Yaskawa INFORM job: A_ROOF_UPPER_0614_2_PAINT_13.JBI

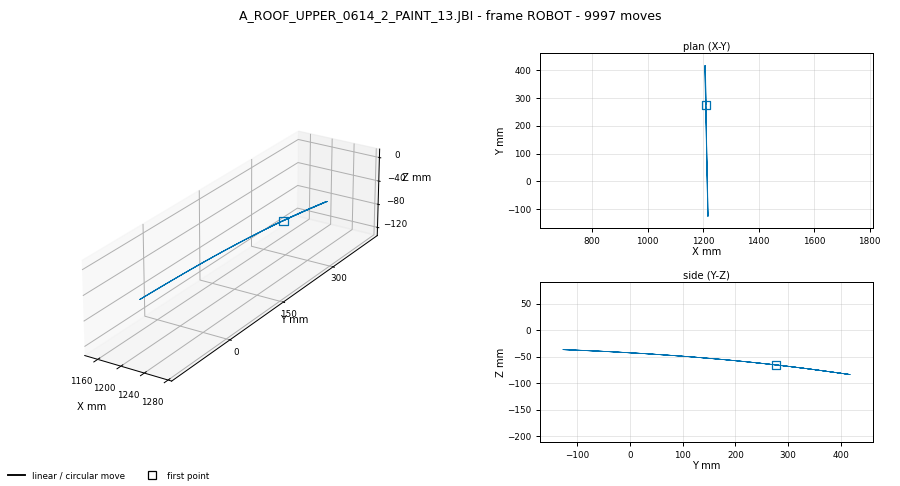
[picture p0: tool path of A_ROOF_UPPER_0614_2_PAINT_13.JBI in frame ROBOT, 9997 of 9997 moves have a stored position in this frame; points joined in program order, loops and branches not executed]
/JOB
//NAME A_ROOF_UPPER_0614_2_PAINT13
//POS
///NPOS 9997,0,0,0,0,0
///TOOL 1
///USER 0
///POSTYPE ROBOT
///RECTAN
///RCONF 1,0,0,0,0,0,0,0,0,0,0,0,0,0,0,0,0,0,0,0,0,0,0,0
C00000=1210.208,276.107,-65.224,-176.767,6.904,148.334
C00001=1210.203,276.355,-65.252,-176.765,6.906,148.334
C00002=1210.199,276.604,-65.280,-176.762,6.909,148.334
C00003=1210.195,276.851,-65.308,-176.760,6.911,148.334
C00004=1210.190,277.100,-65.337,-176.757,6.914,148.333
C00005=1210.186,277.348,-65.365,-176.754,6.916,148.333
C00006=1210.182,277.597,-65.393,-176.752,6.918,148.333
C00007=1210.177,277.845,-65.421,-176.749,6.921,148.333
C00008=1210.173,278.093,-65.449,-176.747,6.923,148.333
C00009=1210.169,278.342,-65.478,-176.744,6.926,148.333
C00010=1210.164,278.590,-65.506,-176.742,6.928,148.333
C00011=1210.160,278.839,-65.535,-176.740,6.930,148.333
C00012=1210.156,279.087,-65.562,-176.737,6.933,148.333
C00013=1210.151,279.335,-65.592,-176.734,6.935,148.332
C00014=1210.147,279.583,-65.620,-176.732,6.938,148.332
C00015=1210.143,279.832,-65.648,-176.729,6.940,148.332
C00016=1210.138,280.080,-65.676,-176.727,6.942,148.332
C00017=1210.134,280.329,-65.705,-176.724,6.945,148.332
C00018=1210.129,280.577,-65.733,-176.722,6.947,148.332
C00019=1210.125,280.826,-65.761,-176.719,6.950,148.332
C00020=1210.121,281.074,-65.790,-176.717,6.952,148.331
C00021=1210.116,281.322,-65.819,-176.715,6.955,148.331
C00022=1210.113,281.570,-65.847,-176.712,6.958,148.331
C00023=1210.107,281.818,-65.875,-176.709,6.959,148.331
C00024=1210.104,282.067,-65.903,-176.707,6.962,148.331
C00025=1210.099,282.316,-65.932,-176.704,6.965,148.331
C00026=1210.094,282.564,-65.961,-176.701,6.967,148.331
C00027=1210.091,282.812,-65.989,-176.699,6.970,148.331
C00028=1210.086,283.060,-66.018,-176.697,6.972,148.331
C00029=1210.082,283.308,-66.047,-176.694,6.975,148.331
C00030=1210.078,283.557,-66.075,-176.692,6.977,148.330
C00031=1210.073,283.805,-66.104,-176.689,6.980,148.330
C00032=1210.069,284.054,-66.132,-176.687,6.982,148.330
C00033=1210.064,284.301,-66.161,-176.685,6.984,148.330
C00034=1210.060,284.550,-66.190,-176.682,6.987,148.330
C00035=1210.056,284.799,-66.218,-176.679,6.989,148.330
C00036=1210.051,285.046,-66.247,-176.677,6.992,148.330
C00037=1210.047,285.295,-66.276,-176.675,6.994,148.330
C00038=1210.043,285.544,-66.304,-176.672,6.997,148.329
C00039=1210.038,285.791,-66.333,-176.669,6.999,148.329
C00040=1210.034,286.040,-66.362,-176.667,7.002,148.329
C00041=1210.030,286.288,-66.390,-176.665,7.004,148.329
C00042=1210.025,286.537,-66.419,-176.662,7.006,148.329
C00043=1210.021,286.785,-66.448,-176.659,7.009,148.329
C00044=1210.016,287.034,-66.477,-176.657,7.011,148.329
C00045=1210.012,287.282,-66.505,-176.654,7.014,148.329
C00046=1210.008,287.530,-66.534,-176.652,7.016,148.329
C00047=1210.003,287.779,-66.563,-176.649,7.019,148.329
C00048=1209.999,288.026,-66.592,-176.647,7.022,148.329
C00049=1209.995,288.275,-66.620,-176.644,7.025,148.329
C00050=1209.991,288.523,-66.650,-176.642,7.027,148.328
C00051=1209.986,288.797,-66.681,-176.639,7.030,148.328
C00052=1209.981,289.071,-66.714,-176.636,7.033,148.328
C00053=1209.977,289.346,-66.745,-176.634,7.036,148.328
C00054=1209.971,289.620,-66.778,-176.631,7.037,148.328
C00055=1209.968,289.868,-66.806,-176.628,7.040,148.328
C00056=1209.963,290.117,-66.835,-176.626,7.043,148.328
C00057=1209.958,290.365,-66.864,-176.624,7.046,148.328
C00058=1209.954,290.613,-66.894,-176.621,7.048,148.328
C00059=1209.950,290.862,-66.922,-176.618,7.051,148.327
C00060=1209.945,291.110,-66.952,-176.616,7.053,148.327
C00061=1209.941,291.357,-66.980,-176.614,7.056,148.327
C00062=1209.937,291.606,-67.009,-176.611,7.058,148.327
C00063=1209.933,291.854,-67.039,-176.609,7.061,148.327
C00064=1209.929,292.103,-67.068,-176.607,7.063,148.327
C00065=1209.924,292.352,-67.097,-176.603,7.066,148.327
C00066=1209.919,292.599,-67.126,-176.601,7.068,148.327
C00067=1209.915,292.847,-67.155,-176.599,7.070,148.327
C00068=1209.911,293.096,-67.184,-176.596,7.073,148.327
C00069=1209.906,293.345,-67.213,-176.594,7.076,148.327
C00070=1209.902,293.593,-67.243,-176.592,7.079,148.327
C00071=1209.897,293.840,-67.272,-176.590,7.081,148.327
C00072=1209.894,294.088,-67.301,-176.586,7.084,148.326
C00073=1209.889,294.337,-67.330,-176.584,7.086,148.326
C00074=1209.885,294.586,-67.359,-176.582,7.089,148.326
C00075=1209.881,294.834,-67.388,-176.579,7.091,148.326
C00076=1209.876,295.081,-67.418,-176.577,7.094,148.326
C00077=1209.872,295.330,-67.447,-176.575,7.096,148.326
C00078=1209.868,295.578,-67.476,-176.572,7.099,148.326
C00079=1209.864,295.826,-67.506,-176.570,7.101,148.326
C00080=1209.859,296.075,-67.535,-176.567,7.104,148.326
C00081=1209.855,296.323,-67.564,-176.565,7.106,148.326
C00082=1209.851,296.572,-67.594,-176.562,7.109,148.326
C00083=1209.847,296.820,-67.623,-176.560,7.112,148.326
C00084=1209.842,297.067,-67.652,-176.557,7.115,148.326
C00085=1209.838,297.316,-67.682,-176.555,7.117,148.326
C00086=1209.834,297.564,-67.711,-176.552,7.120,148.326
C00087=1209.829,297.813,-67.741,-176.550,7.122,148.326
C00088=1209.825,298.061,-67.771,-176.547,7.125,148.326
C00089=1209.820,298.309,-67.800,-176.545,7.127,148.326
C00090=1209.816,298.557,-67.829,-176.543,7.130,148.326
C00091=1209.812,298.806,-67.859,-176.540,7.132,148.325
C00092=1209.808,299.054,-67.888,-176.537,7.135,148.325
C00093=1209.804,299.302,-67.918,-176.535,7.137,148.325
C00094=1209.799,299.550,-67.947,-176.533,7.140,148.325
C00095=1209.795,299.798,-67.976,-176.530,7.143,148.325
C00096=1209.790,300.046,-68.006,-176.528,7.146,148.325
C00097=1209.786,300.295,-68.036,-176.526,7.148,148.325
C00098=1209.782,300.543,-68.066,-176.523,7.151,148.325
C00099=1209.777,300.791,-68.095,-176.521,7.153,148.325
C00100=1209.773,301.039,-68.125,-176.518,7.156,148.325
C00101=1209.769,301.287,-68.154,-176.515,7.159,148.325
C00102=1209.765,301.536,-68.184,-176.513,7.161,148.325
C00103=1209.760,301.784,-68.214,-176.511,7.164,148.325
C00104=1209.756,302.032,-68.243,-176.508,7.167,148.325
C00105=1209.752,302.280,-68.273,-176.506,7.170,148.325
C00106=1209.748,302.528,-68.303,-176.504,7.172,148.325
C00107=1209.743,302.777,-68.333,-176.501,7.175,148.325
C00108=1209.739,303.025,-68.362,-176.499,7.177,148.325
C00109=1209.735,303.273,-68.392,-176.496,7.180,148.325
C00110=1209.731,303.521,-68.422,-176.494,7.182,148.325
C00111=1209.726,303.770,-68.452,-176.491,7.185,148.325
C00112=1209.722,304.018,-68.482,-176.489,7.188,148.324
C00113=1209.718,304.266,-68.512,-176.487,7.191,148.324
C00114=1209.713,304.514,-68.541,-176.484,7.193,148.324
C00115=1209.709,304.762,-68.571,-176.482,7.196,148.324
C00116=1209.704,305.011,-68.601,-176.480,7.198,148.324
C00117=1209.700,305.258,-68.631,-176.477,7.201,148.324
C00118=1209.696,305.507,-68.661,-176.474,7.204,148.324
C00119=1209.692,305.755,-68.691,-176.472,7.206,148.324
C00120=1209.688,306.003,-68.721,-176.469,7.209,148.324
C00121=1209.683,306.251,-68.751,-176.467,7.211,148.324
C00122=1209.679,306.499,-68.781,-176.465,7.215,148.324
C00123=1209.675,306.747,-68.810,-176.463,7.217,148.324
C00124=1209.670,306.995,-68.841,-176.460,7.220,148.324
C00125=1209.666,307.244,-68.870,-176.458,7.222,148.324
C00126=1209.662,307.492,-68.900,-176.456,7.225,148.324
C00127=1209.657,307.740,-68.931,-176.453,7.227,148.324
C00128=1209.653,307.988,-68.960,-176.451,7.231,148.324
C00129=1209.649,308.237,-68.991,-176.448,7.234,148.324
C00130=1209.645,308.485,-69.021,-176.446,7.236,148.324
C00131=1209.641,308.733,-69.051,-176.443,7.239,148.324
C00132=1209.636,308.981,-69.081,-176.441,7.241,148.324
C00133=1209.632,309.229,-69.111,-176.438,7.244,148.324
C00134=1209.627,309.477,-69.141,-176.436,7.246,148.324
C00135=1209.623,309.725,-69.171,-176.434,7.249,148.324
C00136=1209.618,309.973,-69.202,-176.432,7.252,148.324
C00137=1209.614,310.221,-69.232,-176.429,7.255,148.324
C00138=1209.610,310.469,-69.262,-176.427,7.257,148.324
C00139=1209.606,310.718,-69.292,-176.425,7.260,148.324
C00140=1209.602,310.966,-69.322,-176.422,7.263,148.324
C00141=1209.598,311.214,-69.353,-176.420,7.265,148.324
C00142=1209.593,311.462,-69.382,-176.417,7.268,148.324
C00143=1209.589,311.710,-69.413,-176.415,7.271,148.324
C00144=1209.585,311.958,-69.443,-176.413,7.274,148.324
C00145=1209.580,312.206,-69.473,-176.411,7.276,148.324
C00146=1209.577,312.455,-69.504,-176.408,7.279,148.324
C00147=1209.572,312.703,-69.535,-176.406,7.281,148.324
C00148=1209.567,312.951,-69.565,-176.403,7.284,148.324
C00149=1209.563,313.199,-69.595,-176.400,7.287,148.324
C00150=1209.559,313.447,-69.626,-176.399,7.290,148.324
C00151=1209.555,313.696,-69.656,-176.396,7.293,148.324
C00152=1209.551,313.944,-69.686,-176.394,7.295,148.324
C00153=1209.547,314.191,-69.716,-176.391,7.298,148.324
C00154=1209.542,314.439,-69.747,-176.389,7.300,148.324
C00155=1209.537,314.716,-69.781,-176.387,7.303,148.324
C00156=1209.532,314.992,-69.815,-176.384,7.307,148.324
C00157=1209.528,315.268,-69.848,-176.382,7.310,148.324
C00158=1209.524,315.544,-69.883,-176.379,7.313,148.324
C00159=1209.519,315.792,-69.913,-176.376,7.316,148.324
C00160=1209.514,316.040,-69.944,-176.374,7.318,148.324
C00161=1209.511,316.288,-69.974,-176.372,7.321,148.324
C00162=1209.506,316.536,-70.005,-176.369,7.324,148.324
C00163=1209.502,316.785,-70.036,-176.367,7.327,148.324
C00164=1209.498,317.033,-70.066,-176.364,7.330,148.324
C00165=1209.493,317.281,-70.097,-176.362,7.332,148.324
C00166=1209.489,317.529,-70.128,-176.360,7.335,148.325
C00167=1209.485,317.777,-70.158,-176.358,7.337,148.325
C00168=1209.481,318.025,-70.189,-176.355,7.340,148.325
C00169=1209.476,318.273,-70.219,-176.353,7.344,148.325
C00170=1209.473,318.521,-70.250,-176.351,7.346,148.325
C00171=1209.468,318.769,-70.281,-176.348,7.349,148.325
C00172=1209.464,319.017,-70.311,-176.346,7.351,148.325
C00173=1209.459,319.265,-70.342,-176.344,7.355,148.325
C00174=1209.456,319.513,-70.373,-176.342,7.357,148.325
C00175=1209.451,319.761,-70.403,-176.339,7.360,148.325
C00176=1209.446,320.009,-70.434,-176.337,7.363,148.325
C00177=1209.442,320.258,-70.465,-176.335,7.365,148.325
C00178=1209.439,320.506,-70.496,-176.332,7.368,148.325
C00179=1209.434,320.753,-70.527,-176.331,7.371,148.325
C00180=1209.430,321.002,-70.558,-176.328,7.374,148.325
C00181=1209.426,321.249,-70.589,-176.325,7.377,148.325
C00182=1209.422,321.497,-70.619,-176.324,7.380,148.325
C00183=1209.418,321.746,-70.650,-176.321,7.383,148.325
C00184=1209.413,321.994,-70.681,-176.319,7.385,148.325
C00185=1209.408,322.242,-70.712,-176.317,7.388,148.325
C00186=1209.405,322.490,-70.744,-176.314,7.390,148.325
C00187=1209.400,322.738,-70.774,-176.312,7.393,148.325
C00188=1209.396,322.985,-70.805,-176.310,7.397,148.326
C00189=1209.392,323.234,-70.836,-176.307,7.399,148.326
C00190=1209.388,323.482,-70.866,-176.305,7.402,148.326
C00191=1209.384,323.730,-70.898,-176.303,7.404,148.326
C00192=1209.379,323.978,-70.929,-176.300,7.408,148.326
C00193=1209.375,324.226,-70.960,-176.299,7.410,148.326
C00194=1209.371,324.475,-70.991,-176.296,7.413,148.326
C00195=1209.366,324.722,-71.022,-176.293,7.416,148.326
C00196=1209.363,324.970,-71.053,-176.292,7.419,148.326
C00197=1209.359,325.218,-71.084,-176.289,7.422,148.326
C00198=1209.354,325.466,-71.115,-176.287,7.424,148.326
C00199=1209.350,325.714,-71.146,-176.285,7.427,148.326
C00200=1209.346,325.962,-71.177,-176.283,7.431,148.326
C00201=1209.342,326.210,-71.209,-176.280,7.433,148.326
C00202=1209.337,326.458,-71.240,-176.278,7.436,148.326
C00203=1209.333,326.707,-71.271,-176.276,7.438,148.327
C00204=1209.329,326.954,-71.302,-176.273,7.441,148.327
C00205=1209.324,327.202,-71.333,-176.272,7.444,148.327
C00206=1209.321,327.450,-71.365,-176.269,7.447,148.327
C00207=1209.316,327.698,-71.396,-176.267,7.450,148.327
C00208=1209.312,327.947,-71.427,-176.265,7.452,148.327
C00209=1209.308,328.194,-71.458,-176.263,7.456,148.327
C00210=1209.304,328.443,-71.489,-176.260,7.458,148.327
C00211=1209.299,328.690,-71.521,-176.258,7.461,148.327
C00212=1209.295,328.939,-71.552,-176.256,7.464,148.327
C00213=1209.291,329.186,-71.583,-176.254,7.467,148.328
C00214=1209.287,329.435,-71.615,-176.251,7.470,148.328
C00215=1209.283,329.682,-71.646,-176.250,7.472,148.328
C00216=1209.279,329.931,-71.677,-176.247,7.475,148.328
C00217=1209.274,330.178,-71.709,-176.245,7.478,148.328
C00218=1209.270,330.427,-71.740,-176.243,7.481,148.328
C00219=1209.265,330.674,-71.772,-176.240,7.484,148.328
C00220=1209.262,330.922,-71.804,-176.238,7.487,148.328
C00221=1209.257,331.170,-71.835,-176.236,7.490,148.328
C00222=1209.253,331.418,-71.866,-176.234,7.492,148.328
C00223=1209.249,331.666,-71.897,-176.232,7.495,148.328
C00224=1209.245,331.914,-71.929,-176.229,7.499,148.329
C00225=1209.241,332.162,-71.960,-176.227,7.501,148.329
C00226=1209.237,332.410,-71.992,-176.225,7.504,148.329
C00227=1209.232,332.658,-72.024,-176.224,7.507,148.329
C00228=1209.228,332.906,-72.055,-176.221,7.510,148.329
C00229=1209.223,333.154,-72.086,-176.219,7.512,148.329
C00230=1209.220,333.402,-72.118,-176.217,7.515,148.329
C00231=1209.215,333.649,-72.150,-176.214,7.519,148.329
C00232=1209.212,333.898,-72.181,-176.213,7.521,148.330
C00233=1209.207,334.146,-72.213,-176.210,7.524,148.330
C00234=1209.203,334.394,-72.245,-176.208,7.527,148.330
C00235=1209.199,334.642,-72.276,-176.206,7.530,148.330
C00236=1209.195,334.889,-72.308,-176.203,7.533,148.330
C00237=1209.190,335.138,-72.340,-176.202,7.536,148.330
C00238=1209.185,335.386,-72.371,-176.200,7.539,148.330
C00239=1209.182,335.634,-72.403,-176.197,7.541,148.330
C00240=1209.178,335.882,-72.435,-176.195,7.545,148.331
C00241=1209.174,336.129,-72.466,-176.194,7.547,148.331
C00242=1209.169,336.378,-72.498,-176.191,7.550,148.331
C00243=1209.165,336.625,-72.530,-176.189,7.554,148.331
C00244=1209.161,336.873,-72.561,-176.187,7.556,148.331
C00245=1209.157,337.122,-72.594,-176.184,7.559,148.331
C00246=1209.152,337.369,-72.625,-176.183,7.562,148.331
C00247=1209.149,337.617,-72.657,-176.181,7.565,148.332
C00248=1209.145,337.865,-72.689,-176.179,7.568,148.332
C00249=1209.140,338.113,-72.721,-176.176,7.571,148.332
C00250=1209.136,338.361,-72.753,-176.174,7.574,148.332
C00251=1209.132,338.609,-72.784,-176.172,7.576,148.332
C00252=1209.127,338.857,-72.816,-176.170,7.580,148.332
C00253=1209.123,339.105,-72.848,-176.168,7.582,148.332
C00254=1209.119,339.352,-72.879,-176.166,7.585,148.333
C00255=1209.115,339.601,-72.912,-176.164,7.588,148.333
C00256=1209.111,339.849,-72.944,-176.162,7.591,148.333
C00257=1209.106,340.096,-72.976,-176.159,7.594,148.333
C00258=1209.102,340.344,-73.008,-176.158,7.597,148.333
C00259=1209.097,340.622,-73.044,-176.155,7.600,148.333
C00260=1209.093,340.901,-73.080,-176.153,7.603,148.334
C00261=1209.088,341.178,-73.116,-176.151,7.607,148.334
C00262=1209.083,341.457,-73.151,-176.148,7.610,148.334
C00263=1209.079,341.705,-73.183,-176.146,7.613,148.334
C00264=1209.076,341.952,-73.216,-176.144,7.616,148.334
C00265=1209.071,342.201,-73.248,-176.142,7.619,148.334
C00266=1209.067,342.448,-73.280,-176.141,7.622,148.335
C00267=1209.063,342.696,-73.312,-176.138,7.625,148.335
C00268=1209.059,342.944,-73.344,-176.136,7.628,148.335
C00269=1209.054,343.192,-73.376,-176.135,7.631,148.335
C00270=1209.050,343.440,-73.408,-176.132,7.634,148.335
C00271=1209.046,343.688,-73.441,-176.130,7.636,148.335
C00272=1209.042,343.936,-73.473,-176.128,7.640,148.336
C00273=1209.037,344.184,-73.505,-176.126,7.642,148.336
C00274=1209.034,344.432,-73.537,-176.124,7.646,148.336
C00275=1209.029,344.680,-73.569,-176.122,7.649,148.336
C00276=1209.026,344.927,-73.602,-176.120,7.651,148.336
C00277=1209.021,345.175,-73.634,-176.118,7.655,148.337
C00278=1209.017,345.423,-73.666,-176.116,7.657,148.337
C00279=1209.013,345.671,-73.698,-176.114,7.661,148.337
C00280=1209.009,345.919,-73.731,-176.113,7.663,148.337
C00281=1209.004,346.166,-73.763,-176.110,7.666,148.337
C00282=1209.000,346.415,-73.795,-176.109,7.669,148.338
C00283=1208.996,346.662,-73.828,-176.106,7.672,148.338
C00284=1208.992,346.911,-73.860,-176.105,7.675,148.338
C00285=1208.988,347.159,-73.892,-176.103,7.678,148.338
C00286=1208.983,347.406,-73.925,-176.100,7.681,148.339
C00287=1208.979,347.654,-73.957,-176.099,7.684,148.339
C00288=1208.975,347.902,-73.989,-176.097,7.687,148.339
C00289=1208.971,348.150,-74.022,-176.095,7.690,148.339
C00290=1208.967,348.398,-74.054,-176.093,7.693,148.339
C00291=1208.963,348.645,-74.087,-176.091,7.696,148.340
C00292=1208.958,348.893,-74.120,-176.089,7.699,148.340
C00293=1208.954,349.141,-74.151,-176.087,7.702,148.340
C00294=1208.950,349.389,-74.185,-176.085,7.705,148.340
C00295=1208.946,349.637,-74.217,-176.083,7.707,148.340
C00296=1208.942,349.885,-74.250,-176.081,7.711,148.341
C00297=1208.937,350.132,-74.282,-176.079,7.714,148.341
C00298=1208.933,350.380,-74.315,-176.078,7.717,148.341
C00299=1208.930,350.628,-74.347,-176.075,7.720,148.341
C00300=1208.925,350.876,-74.380,-176.074,7.723,148.342
C00301=1208.921,351.124,-74.412,-176.072,7.726,148.342
C00302=1208.918,351.372,-74.445,-176.070,7.729,148.342
C00303=1208.913,351.620,-74.477,-176.068,7.732,148.342
C00304=1208.908,351.867,-74.510,-176.066,7.735,148.342
C00305=1208.904,352.115,-74.543,-176.064,7.738,148.343
C00306=1208.901,352.363,-74.575,-176.063,7.741,148.343
C00307=1208.896,352.610,-74.608,-176.060,7.744,148.343
C00308=1208.892,352.859,-74.641,-176.059,7.747,148.343
C00309=1208.888,353.107,-74.674,-176.057,7.750,148.344
C00310=1208.884,353.354,-74.706,-176.055,7.753,148.344
C00311=1208.880,353.602,-74.739,-176.053,7.756,148.344
C00312=1208.876,353.850,-74.772,-176.052,7.759,148.344
C00313=1208.871,354.098,-74.804,-176.049,7.762,148.345
C00314=1208.867,354.345,-74.837,-176.048,7.765,148.345
C00315=1208.863,354.593,-74.870,-176.046,7.768,148.345
C00316=1208.859,354.841,-74.903,-176.044,7.771,148.345
C00317=1208.855,355.089,-74.935,-176.042,7.774,148.346
C00318=1208.851,355.337,-74.968,-176.041,7.777,148.346
C00319=1208.847,355.584,-75.001,-176.039,7.780,148.346
C00320=1208.843,355.832,-75.033,-176.037,7.783,148.346
C00321=1208.839,356.080,-75.067,-176.035,7.786,148.347
C00322=1208.834,356.328,-75.100,-176.034,7.789,148.347
C00323=1208.830,356.576,-75.133,-176.031,7.792,148.347
C00324=1208.826,356.824,-75.165,-176.030,7.795,148.348
C00325=1208.822,357.072,-75.199,-176.028,7.798,148.348
C00326=1208.818,357.319,-75.231,-176.026,7.801,148.348
C00327=1208.814,357.567,-75.264,-176.025,7.804,148.349
C00328=1208.810,357.815,-75.297,-176.023,7.807,148.349
C00329=1208.806,358.062,-75.331,-176.021,7.810,148.349
C00330=1208.801,358.311,-75.363,-176.019,7.813,148.349
C00331=1208.797,358.558,-75.396,-176.017,7.816,148.350
C00332=1208.793,358.806,-75.429,-176.016,7.819,148.350
C00333=1208.789,359.054,-75.462,-176.014,7.823,148.350
C00334=1208.785,359.302,-75.496,-176.012,7.825,148.350
C00335=1208.781,359.549,-75.529,-176.010,7.829,148.351
C00336=1208.777,359.797,-75.561,-176.009,7.831,148.351
C00337=1208.773,360.044,-75.594,-176.007,7.835,148.351
C00338=1208.769,360.292,-75.628,-176.005,7.837,148.352
C00339=1208.765,360.541,-75.660,-176.004,7.841,148.352
C00340=1208.761,360.788,-75.693,-176.002,7.844,148.352
C00341=1208.756,361.036,-75.726,-176.001,7.846,148.353
C00342=1208.752,361.284,-75.760,-175.999,7.850,148.353
C00343=1208.748,361.531,-75.793,-175.997,7.853,148.353
C00344=1208.744,361.779,-75.826,-175.995,7.856,148.354
C00345=1208.740,362.027,-75.859,-175.994,7.859,148.354
C00346=1208.736,362.275,-75.892,-175.992,7.862,148.354
C00347=1208.732,362.522,-75.925,-175.991,7.865,148.355
C00348=1208.727,362.770,-75.958,-175.989,7.868,148.355
C00349=1208.724,363.017,-75.992,-175.987,7.871,148.355
C00350=1208.719,363.265,-76.026,-175.986,7.874,148.356
C00351=1208.715,363.513,-76.059,-175.984,7.877,148.356
C00352=1208.711,363.760,-76.092,-175.983,7.880,148.356
C00353=1208.707,364.008,-76.125,-175.981,7.883,148.357
C00354=1208.704,364.257,-76.159,-175.979,7.886,148.357
C00355=1208.699,364.505,-76.192,-175.978,7.889,148.357
C00356=1208.694,364.752,-76.225,-175.976,7.893,148.358
C00357=1208.690,365.000,-76.259,-175.975,7.895,148.358
C00358=1208.686,365.248,-76.292,-175.973,7.898,148.358
C00359=1208.682,365.495,-76.326,-175.972,7.902,148.359
C00360=1208.678,365.743,-76.359,-175.970,7.904,148.359
C00361=1208.674,365.990,-76.392,-175.969,7.907,148.359
C00362=1208.670,366.238,-76.425,-175.967,7.911,148.360
C00363=1208.665,366.519,-76.464,-175.965,7.914,148.360
C00364=1208.661,366.799,-76.501,-175.964,7.917,148.360
C00365=1208.656,367.079,-76.538,-175.962,7.920,148.361
C00366=1208.652,367.360,-76.577,-175.960,7.924,148.361
C00367=1208.647,367.608,-76.610,-175.959,7.927,148.362
C00368=1208.644,367.855,-76.644,-175.958,7.930,148.362
C00369=1208.639,368.102,-76.677,-175.956,7.933,148.362
C00370=1208.635,368.350,-76.710,-175.954,7.936,148.363
C00371=1208.631,368.599,-76.744,-175.953,7.939,148.363
C00372=1208.627,368.846,-76.778,-175.951,7.942,148.363
C00373=1208.623,369.094,-76.811,-175.950,7.945,148.364
C00374=1208.619,369.341,-76.844,-175.949,7.948,148.364
C00375=1208.615,369.588,-76.878,-175.948,7.951,148.365
C00376=1208.610,369.837,-76.912,-175.946,7.954,148.365
C00377=1208.607,370.085,-76.946,-175.945,7.957,148.365
C00378=1208.603,370.332,-76.979,-175.943,7.960,148.366
C00379=1208.599,370.580,-77.013,-175.942,7.962,148.366
C00380=1208.594,370.828,-77.046,-175.940,7.966,148.366
C00381=1208.590,371.075,-77.080,-175.939,7.969,148.367
C00382=1208.586,371.323,-77.113,-175.938,7.972,148.367
C00383=1208.582,371.571,-77.147,-175.936,7.975,148.368
C00384=1208.579,371.818,-77.181,-175.935,7.978,148.368
C00385=1208.574,372.066,-77.214,-175.934,7.981,148.368
C00386=1208.570,372.313,-77.248,-175.932,7.984,148.369
C00387=1208.566,372.561,-77.282,-175.931,7.987,148.369
C00388=1208.562,372.809,-77.316,-175.930,7.989,148.370
C00389=1208.558,373.057,-77.350,-175.928,7.993,148.370
C00390=1208.554,373.304,-77.383,-175.927,7.996,148.370
C00391=1208.550,373.552,-77.417,-175.926,7.999,148.371
C00392=1208.545,373.800,-77.450,-175.925,8.002,148.371
C00393=1208.541,374.048,-77.485,-175.923,8.004,148.372
C00394=1208.537,374.295,-77.518,-175.922,8.007,148.372
C00395=1208.533,374.543,-77.552,-175.921,8.010,148.372
C00396=1208.529,374.790,-77.586,-175.920,8.014,148.373
C00397=1208.525,375.038,-77.620,-175.918,8.017,148.373
C00398=1208.521,375.286,-77.654,-175.917,8.020,148.374
C00399=1208.517,375.533,-77.687,-175.916,8.022,148.374
C00400=1208.513,375.781,-77.721,-175.915,8.025,148.375
C00401=1208.509,376.029,-77.755,-175.914,8.028,148.375
C00402=1208.505,376.276,-77.789,-175.912,8.031,148.375
C00403=1208.501,376.524,-77.822,-175.912,8.034,148.376
C00404=1208.496,376.772,-77.857,-175.910,8.037,148.376
C00405=1208.493,377.019,-77.891,-175.909,8.040,148.377
C00406=1208.488,377.267,-77.925,-175.907,8.043,148.377
C00407=1208.484,377.515,-77.958,-175.906,8.046,148.378
C00408=1208.480,377.762,-77.992,-175.906,8.049,148.378
C00409=1208.476,378.010,-78.026,-175.904,8.052,148.379
C00410=1208.472,378.257,-78.060,-175.903,8.055,148.379
C00411=1208.467,378.506,-78.094,-175.902,8.058,148.379
C00412=1208.464,378.753,-78.128,-175.901,8.060,148.380
C00413=1208.460,379.000,-78.162,-175.900,8.063,148.380
C00414=1208.455,379.248,-78.196,-175.899,8.066,148.381
C00415=1208.452,379.496,-78.230,-175.898,8.069,148.381
C00416=1208.448,379.744,-78.265,-175.897,8.072,148.382
C00417=1208.443,379.991,-78.298,-175.896,8.075,148.382
C00418=1208.439,380.239,-78.332,-175.894,8.078,148.383
C00419=1208.436,380.487,-78.367,-175.894,8.081,148.383
C00420=1208.432,380.734,-78.400,-175.892,8.084,148.384
C00421=1208.427,380.982,-78.434,-175.892,8.086,148.384
C00422=1208.424,381.230,-78.468,-175.891,8.089,148.384
C00423=1208.419,381.477,-78.503,-175.890,8.092,148.385
C00424=1208.415,381.724,-78.537,-175.889,8.094,148.385
C00425=1208.411,381.973,-78.571,-175.888,8.098,148.386
C00426=1208.407,382.220,-78.605,-175.887,8.100,148.386
C00427=1208.403,382.467,-78.639,-175.885,8.103,148.387
C00428=1208.399,382.715,-78.673,-175.885,8.106,148.387
C00429=1208.395,382.963,-78.708,-175.883,8.109,148.388
C00430=1208.391,383.210,-78.741,-175.883,8.112,148.388
C00431=1208.387,383.459,-78.776,-175.882,8.114,148.389
C00432=1208.383,383.706,-78.810,-175.881,8.117,148.389
C00433=1208.378,383.953,-78.844,-175.880,8.120,148.390
C00434=1208.375,384.201,-78.878,-175.879,8.123,148.390
C00435=1208.371,384.448,-78.913,-175.878,8.126,148.391
C00436=1208.366,384.696,-78.947,-175.877,8.129,148.391
C00437=1208.362,384.944,-78.981,-175.877,8.131,148.391
C00438=1208.358,385.192,-79.015,-175.875,8.134,148.392
C00439=1208.354,385.439,-79.049,-175.875,8.137,148.392
C00440=1208.350,385.687,-79.084,-175.874,8.140,148.393
C00441=1208.346,385.934,-79.118,-175.873,8.143,148.393
C00442=1208.342,386.182,-79.153,-175.872,8.145,148.394
C00443=1208.338,386.429,-79.187,-175.871,8.148,148.394
C00444=1208.334,386.677,-79.221,-175.870,8.151,148.395
C00445=1208.330,386.925,-79.256,-175.869,8.154,148.395
C00446=1208.326,387.172,-79.289,-175.869,8.156,148.396
C00447=1208.321,387.420,-79.324,-175.868,8.159,148.396
C00448=1208.318,387.668,-79.358,-175.867,8.162,148.397
C00449=1208.313,387.915,-79.392,-175.866,8.165,148.397
C00450=1208.309,388.163,-79.427,-175.865,8.167,148.398
C00451=1208.306,388.410,-79.461,-175.865,8.170,148.398
C00452=1208.301,388.658,-79.495,-175.863,8.173,148.399
C00453=1208.298,388.905,-79.530,-175.863,8.175,148.399
C00454=1208.293,389.153,-79.564,-175.862,8.178,148.400
C00455=1208.289,389.401,-79.599,-175.861,8.181,148.400
C00456=1208.285,389.648,-79.633,-175.861,8.183,148.401
C00457=1208.281,389.896,-79.668,-175.860,8.186,148.401
C00458=1208.277,390.144,-79.702,-175.859,8.189,148.402
C00459=1208.273,390.391,-79.736,-175.859,8.191,148.402
C00460=1208.269,390.639,-79.771,-175.858,8.194,148.403
C00461=1208.264,390.886,-79.805,-175.857,8.196,148.403
C00462=1208.262,391.134,-79.840,-175.856,8.199,148.403
C00463=1208.257,391.381,-79.875,-175.855,8.202,148.404
C00464=1208.253,391.629,-79.910,-175.855,8.205,148.405
C00465=1208.249,391.876,-79.943,-175.854,8.207,148.405
C00466=1208.245,392.124,-79.978,-175.854,8.210,148.406
C00467=1208.240,392.407,-80.017,-175.853,8.213,148.406
C00468=1208.236,392.689,-80.057,-175.852,8.216,148.407
C00469=1208.231,392.972,-80.096,-175.852,8.219,148.407
C00470=1208.226,393.254,-80.135,-175.850,8.222,148.408
C00471=1208.222,393.502,-80.170,-175.850,8.224,148.408
C00472=1208.218,393.749,-80.204,-175.849,8.227,148.409
C00473=1208.214,393.997,-80.239,-175.849,8.229,148.409
C00474=1208.210,394.244,-80.274,-175.848,8.232,148.410
C00475=1208.207,394.491,-80.308,-175.848,8.235,148.410
C00476=1208.202,394.739,-80.343,-175.847,8.237,148.411
C00477=1208.198,394.986,-80.377,-175.846,8.240,148.411
C00478=1208.194,395.234,-80.412,-175.846,8.243,148.412
C00479=1208.190,395.482,-80.446,-175.845,8.245,148.412
C00480=1208.186,395.729,-80.482,-175.844,8.248,148.413
C00481=1208.182,395.976,-80.516,-175.844,8.250,148.413
C00482=1208.178,396.225,-80.551,-175.843,8.253,148.414
C00483=1208.174,396.472,-80.585,-175.843,8.255,148.414
C00484=1208.170,396.720,-80.620,-175.842,8.258,148.415
C00485=1208.166,396.967,-80.655,-175.842,8.261,148.415
C00486=1208.162,397.215,-80.690,-175.841,8.263,148.416
C00487=1208.158,397.462,-80.723,-175.840,8.266,148.416
C00488=1208.154,397.710,-80.758,-175.840,8.268,148.417
C00489=1208.149,397.957,-80.793,-175.839,8.270,148.417
C00490=1208.146,398.205,-80.828,-175.838,8.273,148.418
C00491=1208.141,398.452,-80.863,-175.838,8.275,148.418
C00492=1208.138,398.700,-80.897,-175.837,8.278,148.419
C00493=1208.133,398.948,-80.931,-175.837,8.280,148.419
C00494=1208.130,399.195,-80.967,-175.837,8.283,148.420
C00495=1208.125,399.442,-81.001,-175.836,8.286,148.420
C00496=1208.121,399.691,-81.036,-175.835,8.288,148.421
C00497=1208.118,399.937,-81.071,-175.835,8.290,148.421
C00498=1208.114,400.185,-81.106,-175.834,8.293,148.422
C00499=1208.109,400.433,-81.140,-175.834,8.295,148.422
C00500=1208.105,400.681,-81.175,-175.833,8.297,148.423
C00501=1208.101,400.928,-81.210,-175.833,8.300,148.423
C00502=1208.098,401.175,-81.244,-175.832,8.303,148.424
C00503=1208.093,401.423,-81.279,-175.832,8.305,148.424
C00504=1208.089,401.670,-81.314,-175.832,8.307,148.425
C00505=1208.085,401.918,-81.349,-175.831,8.310,148.425
C00506=1208.081,402.166,-81.384,-175.831,8.312,148.426
C00507=1208.077,402.413,-81.419,-175.830,8.314,148.426
C00508=1208.073,402.661,-81.454,-175.830,8.317,148.427
C00509=1208.070,402.908,-81.489,-175.829,8.320,148.427
C00510=1208.065,403.155,-81.523,-175.828,8.322,148.428
C00511=1208.061,403.403,-81.558,-175.828,8.324,148.428
C00512=1208.057,403.650,-81.593,-175.828,8.326,148.429
C00513=1208.053,403.898,-81.628,-175.828,8.328,148.429
C00514=1208.048,404.146,-81.662,-175.826,8.331,148.430
C00515=1208.045,404.393,-81.698,-175.826,8.334,148.430
C00516=1208.042,404.641,-81.732,-175.826,8.336,148.431
C00517=1208.037,404.888,-81.767,-175.825,8.338,148.431
C00518=1208.033,405.136,-81.802,-175.825,8.340,148.432
C00519=1208.029,405.383,-81.837,-175.825,8.342,148.432
C00520=1208.025,405.631,-81.872,-175.824,8.345,148.433
C00521=1208.021,405.878,-81.907,-175.823,8.347,148.433
C00522=1208.017,406.126,-81.942,-175.823,8.350,148.434
C00523=1208.012,406.373,-81.977,-175.823,8.352,148.434
C00524=1208.009,406.621,-82.012,-175.823,8.354,148.435
C00525=1208.005,406.869,-82.047,-175.822,8.356,148.435
C00526=1208.001,407.115,-82.082,-175.821,8.359,148.436
C00527=1207.997,407.364,-82.117,-175.821,8.362,148.436
C00528=1207.993,407.610,-82.152,-175.820,8.364,148.436
C00529=1207.989,407.858,-82.187,-175.820,8.366,148.437
C00530=1207.985,408.107,-82.221,-175.820,8.368,148.437
C00531=1207.981,408.353,-82.257,-175.820,8.370,148.438
C00532=1207.977,408.601,-82.291,-175.819,8.372,148.438
C00533=1207.972,408.848,-82.327,-175.819,8.375,148.439
C00534=1207.968,409.096,-82.361,-175.819,8.377,148.439
C00535=1207.965,409.344,-82.397,-175.818,8.379,148.440
C00536=1207.960,409.591,-82.431,-175.818,8.381,148.440
C00537=1207.957,409.839,-82.467,-175.817,8.384,148.441
C00538=1207.952,410.086,-82.502,-175.816,8.386,148.441
C00539=1207.948,410.334,-82.537,-175.816,8.388,148.442
C00540=1207.945,410.581,-82.572,-175.816,8.391,148.442
C00541=1207.941,410.828,-82.606,-175.816,8.393,148.443
C00542=1207.937,411.076,-82.642,-175.815,8.395,148.443
C00543=1207.933,411.323,-82.676,-175.815,8.397,148.444
C00544=1207.929,411.571,-82.712,-175.815,8.399,148.444
C00545=1207.925,411.819,-82.747,-175.814,8.401,148.445
C00546=1207.921,412.066,-82.782,-175.814,8.404,148.445
C00547=1207.917,412.314,-82.817,-175.814,8.406,148.446
C00548=1207.912,412.561,-82.852,-175.813,8.408,148.446
C00549=1207.909,412.808,-82.888,-175.813,8.410,148.446
C00550=1207.905,413.056,-82.922,-175.813,8.412,148.447
C00551=1207.901,413.303,-82.958,-175.812,8.414,148.447
C00552=1207.897,413.551,-82.992,-175.812,8.417,148.448
C00553=1207.893,413.799,-83.028,-175.811,8.419,148.448
C00554=1207.889,414.045,-83.063,-175.811,8.421,148.449
C00555=1207.885,414.294,-83.098,-175.811,8.423,148.449
C00556=1207.880,414.540,-83.133,-175.810,8.425,148.450
C00557=1207.877,414.788,-83.168,-175.810,8.427,148.450
C00558=1207.873,415.036,-83.204,-175.809,8.430,148.451
C00559=1207.869,415.283,-83.239,-175.809,8.432,148.451
C00560=1207.865,415.531,-83.274,-175.809,8.434,148.452
C00561=1207.861,415.778,-83.309,-175.808,8.436,148.452
C00562=1207.857,416.025,-83.344,-175.809,8.438,148.453
C00563=1207.852,416.293,-83.383,-175.807,8.440,148.453
C00564=1207.849,416.560,-83.420,-175.807,8.443,148.453
C00565=1207.847,416.827,-83.458,-175.807,8.445,148.454
C00566=1207.849,417.094,-83.495,-175.806,8.447,148.454
C00567=1207.427,417.094,-83.533,-175.810,8.458,148.458
C00568=1207.425,416.825,-83.495,-175.810,8.456,148.458
C00569=1207.427,416.555,-83.457,-175.810,8.453,148.457
C00570=1207.431,416.285,-83.418,-175.811,8.451,148.457
C00571=1207.435,416.015,-83.380,-175.811,8.448,148.456
C00572=1207.438,415.768,-83.344,-175.812,8.446,148.456
C00573=1207.443,415.520,-83.310,-175.812,8.445,148.455
C00574=1207.447,415.273,-83.274,-175.812,8.442,148.455
C00575=1207.450,415.025,-83.239,-175.813,8.440,148.454
C00576=1207.455,414.778,-83.204,-175.813,8.438,148.454
C00577=1207.458,414.530,-83.169,-175.813,8.436,148.453
C00578=1207.463,414.283,-83.134,-175.814,8.434,148.453
C00579=1207.467,414.035,-83.099,-175.814,8.432,148.452
C00580=1207.470,413.788,-83.063,-175.814,8.429,148.452
C00581=1207.475,413.540,-83.029,-175.815,8.427,148.452
C00582=1207.479,413.293,-82.993,-175.815,8.425,148.451
C00583=1207.482,413.045,-82.958,-175.815,8.423,148.451
C00584=1207.487,412.798,-82.923,-175.816,8.421,148.450
C00585=1207.490,412.550,-82.888,-175.816,8.419,148.450
C00586=1207.494,412.302,-82.853,-175.816,8.416,148.449
C00587=1207.499,412.056,-82.818,-175.817,8.414,148.449
C00588=1207.503,411.807,-82.783,-175.817,8.412,148.448
C00589=1207.507,411.561,-82.748,-175.818,8.410,148.448
C00590=1207.511,411.313,-82.712,-175.818,8.408,148.447
C00591=1207.515,411.065,-82.677,-175.818,8.406,148.447
C00592=1207.519,410.818,-82.642,-175.819,8.403,148.446
C00593=1207.523,410.570,-82.607,-175.819,8.401,148.446
C00594=1207.527,410.323,-82.572,-175.820,8.399,148.445
C00595=1207.531,410.075,-82.537,-175.820,8.397,148.445
C00596=1207.535,409.828,-82.502,-175.820,8.395,148.444
C00597=1207.539,409.580,-82.467,-175.821,8.393,148.444
C00598=1207.543,409.333,-82.432,-175.821,8.389,148.443
C00599=1207.547,409.085,-82.397,-175.822,8.387,148.443
C00600=1207.551,408.838,-82.362,-175.822,8.385,148.442
C00601=1207.555,408.590,-82.327,-175.822,8.383,148.442
C00602=1207.559,408.343,-82.292,-175.823,8.381,148.442
C00603=1207.563,408.095,-82.257,-175.823,8.378,148.441
C00604=1207.568,407.848,-82.222,-175.824,8.376,148.441
C00605=1207.572,407.600,-82.187,-175.824,8.374,148.440
C00606=1207.574,407.353,-82.152,-175.824,8.372,148.440
C00607=1207.579,407.105,-82.117,-175.824,8.370,148.439
C00608=1207.583,406.858,-82.082,-175.825,8.368,148.439
C00609=1207.587,406.610,-82.047,-175.826,8.365,148.438
C00610=1207.591,406.363,-82.012,-175.826,8.362,148.438
C00611=1207.595,406.115,-81.977,-175.827,8.360,148.437
C00612=1207.599,405.868,-81.942,-175.827,8.358,148.437
C00613=1207.603,405.620,-81.907,-175.827,8.356,148.436
C00614=1207.607,405.373,-81.872,-175.827,8.353,148.436
C00615=1207.611,405.125,-81.837,-175.828,8.351,148.435
C00616=1207.616,404.877,-81.802,-175.829,8.348,148.435
C00617=1207.619,404.630,-81.768,-175.829,8.346,148.434
C00618=1207.623,404.382,-81.733,-175.829,8.344,148.434
C00619=1207.627,404.135,-81.698,-175.830,8.342,148.433
C00620=1207.631,403.887,-81.663,-175.830,8.340,148.433
C00621=1207.636,403.640,-81.628,-175.831,8.337,148.432
C00622=1207.639,403.392,-81.593,-175.831,8.334,148.432
C00623=1207.644,403.145,-81.558,-175.832,8.332,148.431
C00624=1207.648,402.897,-81.523,-175.832,8.330,148.431
C00625=1207.651,402.650,-81.489,-175.833,8.327,148.430
C00626=1207.655,402.402,-81.454,-175.833,8.325,148.430
C00627=1207.660,402.155,-81.419,-175.833,8.323,148.429
C00628=1207.664,401.907,-81.384,-175.834,8.320,148.429
C00629=1207.668,401.659,-81.349,-175.834,8.317,148.428
C00630=1207.672,401.412,-81.314,-175.835,8.315,148.428
C00631=1207.675,401.165,-81.280,-175.835,8.313,148.427
C00632=1207.680,400.917,-81.245,-175.835,8.311,148.427
C00633=1207.683,400.670,-81.210,-175.836,8.308,148.426
C00634=1207.688,400.422,-81.175,-175.837,8.306,148.426
C00635=1207.692,400.174,-81.140,-175.837,8.303,148.425
C00636=1207.696,399.927,-81.105,-175.838,8.300,148.425
C00637=1207.699,399.679,-81.071,-175.838,8.298,148.424
C00638=1207.704,399.432,-81.036,-175.839,8.296,148.424
C00639=1207.708,399.185,-81.001,-175.840,8.293,148.423
C00640=1207.712,398.937,-80.966,-175.840,8.291,148.423
C00641=1207.716,398.689,-80.932,-175.840,8.289,148.422
C00642=1207.720,398.442,-80.898,-175.841,8.286,148.422
C00643=1207.724,398.194,-80.862,-175.841,8.283,148.421
C00644=1207.728,397.947,-80.828,-175.842,8.281,148.421
C00645=1207.732,397.699,-80.793,-175.843,8.278,148.420
C00646=1207.737,397.451,-80.758,-175.843,8.276,148.420
C00647=1207.740,397.204,-80.724,-175.843,8.274,148.419
C00648=1207.744,396.957,-80.689,-175.844,8.271,148.419
C00649=1207.748,396.709,-80.654,-175.845,8.269,148.418
C00650=1207.753,396.461,-80.620,-175.845,8.266,148.418
C00651=1207.756,396.214,-80.584,-175.846,8.263,148.417
C00652=1207.760,395.967,-80.550,-175.847,8.261,148.417
C00653=1207.764,395.719,-80.515,-175.847,8.258,148.416
C00654=1207.769,395.471,-80.481,-175.847,8.256,148.416
C00655=1207.773,395.223,-80.446,-175.848,8.253,148.415
C00656=1207.777,394.976,-80.412,-175.849,8.251,148.415
C00657=1207.780,394.728,-80.377,-175.849,8.248,148.414
C00658=1207.785,394.481,-80.342,-175.850,8.246,148.414
C00659=1207.788,394.233,-80.308,-175.851,8.243,148.413
C00660=1207.793,393.986,-80.274,-175.851,8.240,148.413
C00661=1207.797,393.738,-80.239,-175.852,8.238,148.412
C00662=1207.801,393.490,-80.204,-175.852,8.235,148.412
C00663=1207.805,393.244,-80.170,-175.853,8.232,148.411
C00664=1207.809,392.961,-80.131,-175.854,8.229,148.411
C00665=1207.814,392.678,-80.091,-175.855,8.226,148.410
C00666=1207.818,392.395,-80.052,-175.855,8.224,148.410
C00667=1207.823,392.114,-80.012,-175.856,8.221,148.409
C00668=1207.827,391.866,-79.977,-175.857,8.218,148.409
C00669=1207.832,391.618,-79.943,-175.858,8.215,148.408
C00670=1207.835,391.370,-79.909,-175.858,8.213,148.408
C00671=1207.839,391.123,-79.874,-175.859,8.210,148.407
C00672=1207.843,390.875,-79.839,-175.860,8.208,148.407
C00673=1207.847,390.628,-79.806,-175.861,8.205,148.406
C00674=1207.852,390.380,-79.771,-175.861,8.201,148.405
C00675=1207.856,390.132,-79.736,-175.862,8.200,148.405
C00676=1207.859,389.885,-79.702,-175.863,8.196,148.405
C00677=1207.863,389.637,-79.668,-175.863,8.194,148.404
C00678=1207.868,389.390,-79.633,-175.864,8.191,148.404
C00679=1207.871,389.142,-79.599,-175.865,8.188,148.403
C00680=1207.876,388.894,-79.564,-175.866,8.186,148.403
C00681=1207.880,388.647,-79.530,-175.866,8.183,148.402
C00682=1207.884,388.399,-79.496,-175.868,8.180,148.402
C00683=1207.888,388.152,-79.461,-175.868,8.178,148.401
C00684=1207.891,387.904,-79.427,-175.868,8.175,148.401
C00685=1207.896,387.656,-79.392,-175.870,8.172,148.400
C00686=1207.901,387.409,-79.358,-175.870,8.169,148.400
C00687=1207.904,387.161,-79.324,-175.871,8.167,148.399
C00688=1207.908,386.914,-79.289,-175.872,8.164,148.399
C00689=1207.912,386.666,-79.255,-175.873,8.161,148.398
C00690=1207.916,386.419,-79.221,-175.874,8.158,148.398
C00691=1207.921,386.171,-79.186,-175.874,8.156,148.397
C00692=1207.924,385.923,-79.152,-175.875,8.153,148.397
C00693=1207.929,385.676,-79.117,-175.876,8.150,148.396
C00694=1207.932,385.429,-79.084,-175.877,8.147,148.396
C00695=1207.936,385.181,-79.049,-175.878,8.144,148.395
C00696=1207.940,384.934,-79.015,-175.879,8.142,148.395
C00697=1207.944,384.685,-78.981,-175.880,8.139,148.394
C00698=1207.948,384.438,-78.947,-175.881,8.136,148.394
C00699=1207.953,384.190,-78.912,-175.882,8.133,148.393
C00700=1207.957,383.942,-78.878,-175.883,8.130,148.393
C00701=1207.961,383.695,-78.844,-175.883,8.128,148.393
C00702=1207.965,383.448,-78.809,-175.884,8.125,148.392
C00703=1207.968,383.200,-78.775,-175.885,8.122,148.392
C00704=1207.973,382.952,-78.741,-175.886,8.119,148.391
C00705=1207.977,382.705,-78.707,-175.887,8.116,148.391
C00706=1207.981,382.457,-78.673,-175.888,8.113,148.390
C00707=1207.985,382.210,-78.639,-175.889,8.110,148.390
C00708=1207.990,381.962,-78.604,-175.890,8.108,148.389
C00709=1207.993,381.714,-78.571,-175.892,8.105,148.389
C00710=1207.998,381.466,-78.536,-175.892,8.102,148.388
C00711=1208.001,381.219,-78.502,-175.893,8.100,148.388
C00712=1208.005,380.971,-78.468,-175.894,8.097,148.387
C00713=1208.010,380.723,-78.434,-175.895,8.094,148.387
C00714=1208.014,380.476,-78.400,-175.896,8.091,148.386
C00715=1208.017,380.228,-78.366,-175.897,8.088,148.386
C00716=1208.021,379.981,-78.332,-175.898,8.085,148.386
C00717=1208.026,379.733,-78.298,-175.899,8.082,148.385
C00718=1208.029,379.485,-78.264,-175.900,8.079,148.385
C00719=1208.034,379.238,-78.229,-175.901,8.076,148.384
C00720=1208.038,378.990,-78.196,-175.902,8.074,148.384
C00721=1208.043,378.743,-78.162,-175.904,8.071,148.383
C00722=1208.046,378.495,-78.127,-175.905,8.068,148.383
C00723=1208.051,378.247,-78.094,-175.906,8.065,148.382
C00724=1208.055,378.000,-78.060,-175.907,8.062,148.382
C00725=1208.058,377.752,-78.026,-175.908,8.059,148.382
C00726=1208.063,377.504,-77.992,-175.909,8.056,148.381
C00727=1208.066,377.257,-77.958,-175.910,8.053,148.381
C00728=1208.071,377.009,-77.924,-175.911,8.050,148.380
C00729=1208.075,376.761,-77.890,-175.912,8.048,148.380
C00730=1208.078,376.514,-77.856,-175.914,8.044,148.379
C00731=1208.083,376.266,-77.822,-175.915,8.041,148.379
C00732=1208.087,376.018,-77.789,-175.916,8.038,148.378
C00733=1208.090,375.771,-77.754,-175.917,8.035,148.378
C00734=1208.095,375.523,-77.721,-175.919,8.032,148.378
C00735=1208.099,375.276,-77.687,-175.920,8.030,148.377
C00736=1208.103,375.028,-77.654,-175.921,8.027,148.377
C00737=1208.107,374.780,-77.619,-175.922,8.024,148.376
C00738=1208.111,374.532,-77.586,-175.923,8.021,148.376
C00739=1208.115,374.285,-77.552,-175.925,8.018,148.376
C00740=1208.120,374.037,-77.518,-175.926,8.015,148.375
C00741=1208.123,373.789,-77.484,-175.927,8.012,148.375
C00742=1208.127,373.541,-77.450,-175.928,8.009,148.374
C00743=1208.132,373.294,-77.416,-175.929,8.006,148.374
C00744=1208.136,373.046,-77.383,-175.931,8.003,148.373
C00745=1208.140,372.799,-77.349,-175.932,8.000,148.373
C00746=1208.143,372.551,-77.315,-175.934,7.997,148.373
C00747=1208.148,372.303,-77.281,-175.935,7.994,148.372
C00748=1208.152,372.055,-77.248,-175.936,7.991,148.372
C00749=1208.156,371.808,-77.214,-175.937,7.988,148.371
C00750=1208.160,371.560,-77.180,-175.939,7.985,148.371
C00751=1208.164,371.312,-77.147,-175.940,7.982,148.371
C00752=1208.168,371.065,-77.113,-175.941,7.979,148.370
C00753=1208.172,370.817,-77.080,-175.943,7.976,148.370
C00754=1208.177,370.570,-77.045,-175.944,7.973,148.369
C00755=1208.181,370.322,-77.012,-175.946,7.970,148.369
C00756=1208.185,370.073,-76.979,-175.947,7.967,148.369
C00757=1208.188,369.826,-76.945,-175.948,7.964,148.368
C00758=1208.193,369.579,-76.912,-175.950,7.961,148.368
C00759=1208.197,369.331,-76.878,-175.951,7.958,148.368
C00760=1208.201,369.083,-76.844,-175.953,7.955,148.367
C00761=1208.205,368.836,-76.811,-175.954,7.952,148.367
C00762=1208.209,368.587,-76.777,-175.956,7.949,148.366
C00763=1208.213,368.340,-76.743,-175.957,7.946,148.366
C00764=1208.218,368.092,-76.710,-175.958,7.943,148.366
C00765=1208.222,367.844,-76.676,-175.960,7.940,148.365
C00766=1208.226,367.597,-76.643,-175.961,7.937,148.365
C00767=1208.230,367.350,-76.609,-175.963,7.934,148.365
C00768=1208.235,367.068,-76.572,-175.964,7.930,148.364
C00769=1208.239,366.788,-76.534,-175.967,7.927,148.364
C00770=1208.243,366.508,-76.496,-175.968,7.923,148.363
C00771=1208.248,366.228,-76.458,-175.969,7.921,148.363
C00772=1208.252,365.980,-76.425,-175.971,7.917,148.363
C00773=1208.256,365.732,-76.391,-175.972,7.914,148.362
C00774=1208.261,365.485,-76.358,-175.974,7.912,148.362
C00775=1208.265,365.237,-76.325,-175.976,7.908,148.362
C00776=1208.269,364.989,-76.292,-175.977,7.905,148.361
C00777=1208.272,364.741,-76.258,-175.979,7.902,148.361
C00778=1208.276,364.494,-76.225,-175.980,7.899,148.361
C00779=1208.281,364.246,-76.191,-175.982,7.896,148.360
C00780=1208.285,363.998,-76.158,-175.984,7.893,148.360
C00781=1208.289,363.750,-76.124,-175.985,7.890,148.360
C00782=1208.294,363.502,-76.091,-175.987,7.886,148.359
C00783=1208.298,363.255,-76.058,-175.989,7.884,148.359
C00784=1208.302,363.007,-76.025,-175.990,7.881,148.359
C00785=1208.306,362.759,-75.992,-175.992,7.878,148.358
C00786=1208.310,362.512,-75.959,-175.993,7.875,148.358
C00787=1208.314,362.264,-75.926,-175.995,7.871,148.357
C00788=1208.318,362.017,-75.892,-175.997,7.869,148.357
C00789=1208.322,361.769,-75.859,-175.998,7.865,148.357
C00790=1208.326,361.521,-75.825,-176.000,7.863,148.357
C00791=1208.330,361.273,-75.792,-176.001,7.860,148.356
C00792=1208.334,361.025,-75.759,-176.003,7.857,148.356
C00793=1208.338,360.777,-75.726,-176.005,7.854,148.356
C00794=1208.343,360.529,-75.693,-176.007,7.850,148.355
C00795=1208.347,360.281,-75.660,-176.008,7.848,148.355
C00796=1208.351,360.034,-75.627,-176.010,7.844,148.355
C00797=1208.355,359.786,-75.594,-176.011,7.841,148.354
C00798=1208.359,359.538,-75.560,-176.014,7.838,148.354
C00799=1208.363,359.290,-75.527,-176.015,7.835,148.354
C00800=1208.367,359.043,-75.495,-176.017,7.832,148.354
C00801=1208.371,358.795,-75.462,-176.018,7.829,148.353
C00802=1208.375,358.547,-75.428,-176.020,7.826,148.353
C00803=1208.379,358.300,-75.395,-176.022,7.823,148.353
C00804=1208.383,358.052,-75.362,-176.024,7.820,148.352
C00805=1208.388,357.804,-75.330,-176.025,7.817,148.352
C00806=1208.392,357.556,-75.297,-176.027,7.813,148.352
C00807=1208.396,357.308,-75.263,-176.029,7.811,148.352
C00808=1208.400,357.060,-75.230,-176.031,7.808,148.351
C00809=1208.404,356.813,-75.197,-176.032,7.805,148.351
C00810=1208.408,356.565,-75.165,-176.034,7.801,148.351
C00811=1208.412,356.317,-75.132,-176.036,7.799,148.350
C00812=1208.416,356.069,-75.099,-176.038,7.795,148.350
C00813=1208.421,355.822,-75.066,-176.040,7.793,148.350
C00814=1208.425,355.574,-75.034,-176.042,7.789,148.350
C00815=1208.430,355.326,-75.001,-176.043,7.787,148.349
C00816=1208.433,355.079,-74.968,-176.045,7.783,148.349
C00817=1208.437,354.831,-74.935,-176.047,7.781,148.349
C00818=1208.441,354.583,-74.902,-176.049,7.777,148.349
C00819=1208.446,354.335,-74.869,-176.050,7.775,148.348
C00820=1208.450,354.087,-74.836,-176.052,7.771,148.348
C00821=1208.453,353.839,-74.804,-176.054,7.769,148.348
C00822=1208.458,353.591,-74.771,-176.056,7.765,148.348
C00823=1208.462,353.344,-74.738,-176.058,7.763,148.347
C00824=1208.466,353.095,-74.705,-176.060,7.759,148.347
C00825=1208.470,352.848,-74.673,-176.061,7.757,148.347
C00826=1208.474,352.601,-74.640,-176.064,7.753,148.347
C00827=1208.479,352.353,-74.608,-176.065,7.751,148.346
C00828=1208.483,352.105,-74.575,-176.067,7.747,148.346
C00829=1208.487,351.857,-74.543,-176.069,7.745,148.346
C00830=1208.491,351.609,-74.510,-176.071,7.741,148.346
C00831=1208.495,351.361,-74.477,-176.073,7.739,148.345
C00832=1208.499,351.113,-74.444,-176.075,7.735,148.345
C00833=1208.503,350.866,-74.411,-176.077,7.732,148.345
C00834=1208.508,350.618,-74.379,-176.079,7.730,148.345
C00835=1208.512,350.370,-74.346,-176.080,7.726,148.344
C00836=1208.516,350.122,-74.314,-176.082,7.723,148.344
C00837=1208.520,349.874,-74.281,-176.084,7.720,148.344
C00838=1208.524,349.626,-74.249,-176.086,7.718,148.344
C00839=1208.528,349.378,-74.217,-176.088,7.714,148.343
C00840=1208.532,349.130,-74.184,-176.090,7.712,148.343
C00841=1208.537,348.883,-74.152,-176.092,7.708,148.343
C00842=1208.541,348.635,-74.119,-176.094,7.706,148.343
C00843=1208.545,348.387,-74.087,-176.096,7.702,148.343
C00844=1208.549,348.139,-74.053,-176.098,7.699,148.342
C00845=1208.553,347.891,-74.022,-176.100,7.697,148.342
C00846=1208.558,347.643,-73.990,-176.102,7.693,148.342
C00847=1208.561,347.396,-73.957,-176.104,7.691,148.342
C00848=1208.566,347.148,-73.925,-176.106,7.687,148.342
C00849=1208.570,346.900,-73.891,-176.107,7.685,148.341
C00850=1208.574,346.652,-73.860,-176.110,7.682,148.341
C00851=1208.579,346.404,-73.827,-176.111,7.679,148.341
C00852=1208.582,346.156,-73.796,-176.113,7.676,148.341
C00853=1208.586,345.908,-73.762,-176.115,7.673,148.341
C00854=1208.591,345.660,-73.730,-176.117,7.670,148.340
C00855=1208.595,345.412,-73.698,-176.120,7.667,148.340
C00856=1208.599,345.165,-73.665,-176.121,7.664,148.340
C00857=1208.603,344.917,-73.634,-176.123,7.661,148.340
C00858=1208.607,344.669,-73.601,-176.125,7.658,148.340
C00859=1208.611,344.421,-73.569,-176.127,7.655,148.339
C00860=1208.616,344.174,-73.536,-176.129,7.652,148.339
C00861=1208.620,343.926,-73.505,-176.131,7.649,148.339
C00862=1208.624,343.677,-73.472,-176.133,7.646,148.339
C00863=1208.628,343.430,-73.441,-176.135,7.643,148.339
C00864=1208.633,343.182,-73.408,-176.137,7.640,148.338
C00865=1208.636,342.934,-73.376,-176.139,7.637,148.338
C00866=1208.641,342.686,-73.343,-176.142,7.634,148.338
C00867=1208.645,342.438,-73.312,-176.143,7.632,148.338
C00868=1208.649,342.190,-73.279,-176.145,7.628,148.338
C00869=1208.653,341.942,-73.247,-176.148,7.625,148.338
C00870=1208.658,341.694,-73.215,-176.149,7.622,148.337
C00871=1208.662,341.446,-73.184,-176.151,7.619,148.337
C00872=1208.666,341.168,-73.147,-176.154,7.616,148.337
C00873=1208.671,340.890,-73.111,-176.156,7.613,148.337
C00874=1208.676,340.612,-73.076,-176.159,7.609,148.337
C00875=1208.680,340.333,-73.039,-176.161,7.606,148.336
C00876=1208.685,340.086,-73.008,-176.162,7.604,148.336
C00877=1208.688,339.838,-72.976,-176.165,7.600,148.336
C00878=1208.693,339.590,-72.944,-176.167,7.598,148.336
C00879=1208.697,339.342,-72.912,-176.169,7.595,148.336
C00880=1208.701,339.094,-72.880,-176.171,7.591,148.336
C00881=1208.705,338.846,-72.848,-176.173,7.589,148.335
C00882=1208.710,338.598,-72.816,-176.176,7.586,148.335
C00883=1208.714,338.350,-72.784,-176.177,7.583,148.335
C00884=1208.718,338.103,-72.752,-176.179,7.580,148.335
C00885=1208.722,337.855,-72.721,-176.182,7.577,148.335
C00886=1208.726,337.607,-72.689,-176.184,7.574,148.335
C00887=1208.731,337.359,-72.657,-176.186,7.571,148.335
C00888=1208.735,337.111,-72.625,-176.188,7.568,148.334
C00889=1208.738,336.863,-72.593,-176.190,7.565,148.334
C00890=1208.743,336.615,-72.561,-176.192,7.563,148.334
C00891=1208.747,336.367,-72.530,-176.194,7.560,148.334
C00892=1208.751,336.119,-72.498,-176.196,7.556,148.334
C00893=1208.755,335.871,-72.466,-176.198,7.554,148.334
C00894=1208.760,335.623,-72.434,-176.201,7.551,148.334
C00895=1208.764,335.376,-72.402,-176.202,7.548,148.334
C00896=1208.768,335.128,-72.371,-176.205,7.545,148.333
C00897=1208.772,334.880,-72.340,-176.207,7.542,148.333
C00898=1208.777,334.631,-72.307,-176.209,7.539,148.333
C00899=1208.781,334.383,-72.276,-176.212,7.536,148.333
C00900=1208.785,334.136,-72.244,-176.213,7.534,148.333
C00901=1208.789,333.887,-72.213,-176.215,7.530,148.333
C00902=1208.793,333.640,-72.182,-176.217,7.528,148.333
C00903=1208.798,333.392,-72.149,-176.220,7.525,148.333
C00904=1208.802,333.144,-72.118,-176.222,7.522,148.333
C00905=1208.806,332.896,-72.086,-176.224,7.519,148.332
C00906=1208.810,332.647,-72.055,-176.226,7.516,148.332
C00907=1208.814,332.400,-72.023,-176.228,7.514,148.332
C00908=1208.818,332.152,-71.992,-176.231,7.510,148.332
C00909=1208.823,331.904,-71.960,-176.233,7.507,148.332
C00910=1208.827,331.655,-71.929,-176.235,7.505,148.332
C00911=1208.831,331.408,-71.897,-176.237,7.501,148.332
C00912=1208.835,331.160,-71.865,-176.239,7.499,148.332
C00913=1208.840,330.912,-71.835,-176.241,7.496,148.331
C00914=1208.843,330.664,-71.803,-176.244,7.493,148.331
C00915=1208.848,330.416,-71.772,-176.246,7.490,148.331
C00916=1208.852,330.168,-71.740,-176.248,7.487,148.331
C00917=1208.856,329.920,-71.709,-176.250,7.485,148.331
C00918=1208.861,329.672,-71.677,-176.253,7.482,148.331
C00919=1208.865,329.424,-71.646,-176.254,7.479,148.331
C00920=1208.869,329.176,-71.614,-176.257,7.476,148.331
C00921=1208.873,328.928,-71.583,-176.259,7.473,148.331
C00922=1208.877,328.680,-71.552,-176.261,7.470,148.330
C00923=1208.882,328.432,-71.520,-176.264,7.467,148.330
C00924=1208.886,328.184,-71.489,-176.265,7.465,148.330
C00925=1208.890,327.936,-71.458,-176.268,7.462,148.330
C00926=1208.894,327.688,-71.427,-176.270,7.458,148.330
C00927=1208.899,327.440,-71.396,-176.272,7.456,148.330
C00928=1208.903,327.192,-71.364,-176.275,7.453,148.330
C00929=1208.907,326.944,-71.333,-176.277,7.451,148.330
C00930=1208.911,326.696,-71.302,-176.279,7.448,148.330
C00931=1208.915,326.448,-71.271,-176.282,7.444,148.330
C00932=1208.920,326.200,-71.240,-176.284,7.442,148.330
C00933=1208.924,325.952,-71.208,-176.286,7.439,148.330
C00934=1208.928,325.704,-71.177,-176.288,7.437,148.330
C00935=1208.933,325.456,-71.146,-176.290,7.433,148.329
C00936=1208.936,325.208,-71.115,-176.292,7.431,148.329
C00937=1208.940,324.960,-71.084,-176.295,7.428,148.329
C00938=1208.944,324.711,-71.053,-176.297,7.425,148.329
C00939=1208.949,324.464,-71.022,-176.299,7.422,148.329
C00940=1208.953,324.216,-70.991,-176.301,7.419,148.329
C00941=1208.957,323.967,-70.960,-176.304,7.417,148.329
C00942=1208.962,323.720,-70.929,-176.306,7.414,148.329
C00943=1208.966,323.471,-70.897,-176.309,7.410,148.329
C00944=1208.970,323.223,-70.867,-176.311,7.408,148.329
C00945=1208.974,322.976,-70.836,-176.313,7.405,148.329
C00946=1208.978,322.727,-70.805,-176.315,7.403,148.329
C00947=1208.983,322.480,-70.774,-176.318,7.400,148.329
C00948=1208.987,322.231,-70.743,-176.320,7.396,148.329
C00949=1208.991,321.983,-70.712,-176.322,7.394,148.329
C00950=1208.996,321.735,-70.681,-176.325,7.391,148.329
C00951=1208.999,321.487,-70.651,-176.326,7.389,148.328
C00952=1209.004,321.239,-70.620,-176.329,7.386,148.328
C00953=1209.008,320.992,-70.588,-176.331,7.383,148.328
C00954=1209.012,320.743,-70.557,-176.333,7.380,148.328
C00955=1209.017,320.495,-70.527,-176.336,7.377,148.328
C00956=1209.020,320.247,-70.496,-176.338,7.375,148.328
C00957=1209.024,319.999,-70.465,-176.340,7.371,148.328
C00958=1209.029,319.751,-70.434,-176.342,7.369,148.328
C00959=1209.034,319.503,-70.404,-176.345,7.366,148.328
C00960=1209.038,319.255,-70.374,-176.347,7.363,148.328
C00961=1209.042,319.006,-70.342,-176.349,7.361,148.328
C00962=1209.046,318.758,-70.312,-176.352,7.358,148.328
C00963=1209.051,318.510,-70.281,-176.354,7.355,148.328
C00964=1209.054,318.262,-70.250,-176.356,7.352,148.328
C00965=1209.059,318.014,-70.220,-176.359,7.350,148.328
C00966=1209.063,317.766,-70.189,-176.361,7.347,148.328
C00967=1209.067,317.519,-70.159,-176.363,7.343,148.328
C00968=1209.071,317.270,-70.127,-176.366,7.341,148.328
C00969=1209.076,317.022,-70.097,-176.368,7.338,148.328
C00970=1209.080,316.774,-70.067,-176.370,7.336,148.328
C00971=1209.084,316.526,-70.036,-176.373,7.333,148.328
C00972=1209.088,316.278,-70.005,-176.375,7.330,148.328
C00973=1209.092,316.030,-69.974,-176.377,7.327,148.328
C00974=1209.097,315.781,-69.944,-176.380,7.324,148.328
C00975=1209.102,315.534,-69.914,-176.382,7.322,148.328
C00976=1209.106,315.257,-69.879,-176.384,7.319,148.327
C00977=1209.110,314.981,-69.846,-176.387,7.316,148.327
C00978=1209.115,314.705,-69.812,-176.390,7.313,148.327
C00979=1209.120,314.429,-69.778,-176.392,7.310,148.327
C00980=1209.125,314.181,-69.747,-176.395,7.307,148.327
C00981=1209.129,313.933,-69.717,-176.397,7.304,148.328
C00982=1209.133,313.685,-69.687,-176.399,7.301,148.327
C00983=1209.136,313.437,-69.656,-176.402,7.299,148.327
C00984=1209.141,313.188,-69.626,-176.404,7.296,148.327
C00985=1209.146,312.940,-69.595,-176.407,7.293,148.327
C00986=1209.150,312.693,-69.565,-176.409,7.291,148.327
C00987=1209.154,312.445,-69.534,-176.412,7.288,148.327
C00988=1209.158,312.196,-69.504,-176.413,7.285,148.327
C00989=1209.163,311.948,-69.474,-176.416,7.282,148.327
C00990=1209.167,311.700,-69.443,-176.418,7.280,148.327
C00991=1209.171,311.452,-69.413,-176.421,7.277,148.327
C00992=1209.175,311.204,-69.383,-176.423,7.275,148.327
C00993=1209.180,310.956,-69.353,-176.426,7.272,148.327
C00994=1209.184,310.708,-69.323,-176.428,7.269,148.327
C00995=1209.188,310.459,-69.292,-176.430,7.266,148.327
C00996=1209.192,310.211,-69.262,-176.433,7.263,148.327
C00997=1209.197,309.963,-69.232,-176.435,7.261,148.327
C00998=1209.201,309.715,-69.202,-176.437,7.258,148.327
C00999=1209.205,309.467,-69.172,-176.440,7.256,148.327
C01000=1209.210,309.219,-69.141,-176.442,7.253,148.327
C01001=1209.214,308.971,-69.112,-176.445,7.250,148.327
C01002=1209.218,308.723,-69.081,-176.447,7.247,148.327
C01003=1209.223,308.474,-69.052,-176.450,7.244,148.327
C01004=1209.227,308.226,-69.021,-176.451,7.242,148.327
C01005=1209.231,307.977,-68.991,-176.454,7.239,148.327
C01006=1209.235,307.730,-68.961,-176.456,7.237,148.327
C01007=1209.240,307.481,-68.931,-176.459,7.234,148.327
C01008=1209.243,307.234,-68.901,-176.461,7.231,148.327
C01009=1209.248,306.985,-68.871,-176.464,7.228,148.327
C01010=1209.253,306.737,-68.841,-176.466,7.225,148.327
C01011=1209.256,306.489,-68.811,-176.469,7.223,148.327
C01012=1209.261,306.241,-68.781,-176.471,7.220,148.327
C01013=1209.265,305.993,-68.751,-176.473,7.218,148.328
C01014=1209.269,305.745,-68.721,-176.476,7.215,148.328
C01015=1209.274,305.496,-68.691,-176.478,7.213,148.328
C01016=1209.278,305.248,-68.661,-176.481,7.210,148.328
C01017=1209.282,305.000,-68.632,-176.483,7.207,148.328
C01018=1209.287,304.752,-68.602,-176.486,7.204,148.328
C01019=1209.291,304.504,-68.571,-176.488,7.202,148.328
C01020=1209.295,304.256,-68.542,-176.490,7.199,148.328
C01021=1209.300,304.007,-68.513,-176.493,7.197,148.328
C01022=1209.304,303.759,-68.482,-176.495,7.194,148.328
C01023=1209.308,303.511,-68.452,-176.498,7.191,148.328
C01024=1209.313,303.263,-68.423,-176.500,7.188,148.328
C01025=1209.317,303.015,-68.393,-176.502,7.185,148.328
C01026=1209.321,302.767,-68.363,-176.504,7.183,148.328
C01027=1209.326,302.518,-68.333,-176.507,7.180,148.328
C01028=1209.330,302.270,-68.304,-176.510,7.178,148.328
C01029=1209.334,302.022,-68.274,-176.512,7.175,148.328
C01030=1209.339,301.773,-68.244,-176.514,7.173,148.328
C01031=1209.343,301.526,-68.214,-176.517,7.170,148.328
C01032=1209.347,301.277,-68.185,-176.519,7.168,148.328
C01033=1209.351,301.029,-68.155,-176.522,7.165,148.328
C01034=1209.355,300.781,-68.126,-176.524,7.162,148.328
C01035=1209.359,300.533,-68.096,-176.527,7.159,148.328
C01036=1209.364,300.284,-68.066,-176.529,7.157,148.328
C01037=1209.368,300.036,-68.037,-176.532,7.154,148.328
C01038=1209.373,299.787,-68.007,-176.534,7.152,148.328
C01039=1209.377,299.540,-67.977,-176.536,7.149,148.328
C01040=1209.381,299.292,-67.948,-176.539,7.146,148.328
C01041=1209.385,299.043,-67.918,-176.541,7.144,148.329
C01042=1209.390,298.796,-67.889,-176.544,7.141,148.329
C01043=1209.394,298.547,-67.860,-176.546,7.139,148.329
C01044=1209.399,298.299,-67.830,-176.549,7.136,148.329
C01045=1209.403,298.051,-67.800,-176.551,7.133,148.329
C01046=1209.407,297.802,-67.771,-176.553,7.130,148.329
C01047=1209.411,297.554,-67.741,-176.556,7.128,148.329
C01048=1209.416,297.306,-67.712,-176.558,7.125,148.329
C01049=1209.420,297.057,-67.682,-176.561,7.123,148.329
C01050=1209.424,296.809,-67.653,-176.564,7.120,148.329
C01051=1209.428,296.561,-67.623,-176.566,7.118,148.329
C01052=1209.433,296.313,-67.595,-176.568,7.115,148.329
C01053=1209.437,296.065,-67.566,-176.570,7.113,148.329
C01054=1209.442,295.816,-67.536,-176.573,7.110,148.329
C01055=1209.446,295.568,-67.507,-176.575,7.107,148.329
C01056=1209.450,295.320,-67.477,-176.578,7.104,148.329
C01057=1209.454,295.071,-67.448,-176.580,7.102,148.329
C01058=1209.458,294.823,-67.418,-176.583,7.099,148.329
C01059=1209.463,294.576,-67.389,-176.585,7.097,148.330
C01060=1209.468,294.327,-67.361,-176.588,7.094,148.330
C01061=1209.472,294.078,-67.331,-176.590,7.092,148.330
C01062=1209.476,293.830,-67.302,-176.593,7.089,148.330
C01063=1209.480,293.582,-67.272,-176.595,7.087,148.330
C01064=1209.485,293.334,-67.243,-176.598,7.084,148.330
C01065=1209.489,293.085,-67.214,-176.600,7.082,148.330
C01066=1209.494,292.837,-67.185,-176.603,7.079,148.330
C01067=1209.497,292.589,-67.156,-176.605,7.077,148.330
C01068=1209.501,292.341,-67.127,-176.608,7.074,148.330
C01069=1209.506,292.093,-67.098,-176.610,7.072,148.330
C01070=1209.510,291.845,-67.069,-176.612,7.069,148.330
C01071=1209.515,291.596,-67.039,-176.615,7.066,148.330
C01072=1209.519,291.347,-67.011,-176.617,7.064,148.330
C01073=1209.523,291.099,-66.981,-176.620,7.061,148.331
C01074=1209.528,290.852,-66.952,-176.622,7.059,148.331
C01075=1209.532,290.603,-66.924,-176.625,7.056,148.331
C01076=1209.536,290.355,-66.894,-176.627,7.054,148.331
C01077=1209.540,290.106,-66.865,-176.630,7.051,148.331
C01078=1209.545,289.858,-66.837,-176.632,7.049,148.331
C01079=1209.549,289.610,-66.807,-176.635,7.046,148.331
C01080=1209.554,289.336,-66.776,-176.638,7.043,148.331
C01081=1209.559,289.061,-66.744,-176.640,7.041,148.331
C01082=1209.564,288.788,-66.712,-176.643,7.038,148.331
C01083=1209.568,288.513,-66.680,-176.646,7.035,148.332
C01084=1209.573,288.264,-66.651,-176.648,7.032,148.332
C01085=1209.577,288.016,-66.622,-176.650,7.030,148.332
C01086=1209.582,287.768,-66.593,-176.653,7.028,148.332
C01087=1209.586,287.520,-66.564,-176.656,7.025,148.332
C01088=1209.590,287.271,-66.536,-176.658,7.023,148.332
C01089=1209.594,287.023,-66.506,-176.661,7.020,148.332
C01090=1209.599,286.775,-66.478,-176.663,7.018,148.332
C01091=1209.603,286.527,-66.449,-176.666,7.015,148.332
C01092=1209.607,286.278,-66.420,-176.668,7.013,148.332
C01093=1209.612,286.030,-66.391,-176.671,7.010,148.332
C01094=1209.616,285.782,-66.363,-176.673,7.007,148.332
C01095=1209.620,285.533,-66.334,-176.676,7.005,148.333
C01096=1209.625,285.285,-66.305,-176.678,7.002,148.333
C01097=1209.629,285.036,-66.277,-176.680,7.000,148.333
C01098=1209.633,284.788,-66.248,-176.683,6.997,148.333
C01099=1209.638,284.540,-66.219,-176.685,6.995,148.333
C01100=1209.642,284.291,-66.191,-176.688,6.992,148.333
C01101=1209.647,284.044,-66.162,-176.690,6.990,148.333
C01102=1209.651,283.795,-66.133,-176.693,6.987,148.333
C01103=1209.655,283.546,-66.105,-176.696,6.985,148.334
C01104=1209.660,283.298,-66.077,-176.698,6.983,148.334
C01105=1209.664,283.050,-66.047,-176.700,6.980,148.334
C01106=1209.668,282.801,-66.019,-176.703,6.978,148.334
C01107=1209.673,282.553,-65.991,-176.706,6.975,148.334
C01108=1209.676,282.305,-65.962,-176.708,6.973,148.334
C01109=1209.681,282.057,-65.934,-176.711,6.970,148.334
C01110=1209.686,281.808,-65.905,-176.713,6.968,148.334
C01111=1209.690,281.560,-65.877,-176.715,6.966,148.334
C01112=1209.695,281.311,-65.848,-176.718,6.963,148.334
C01113=1209.698,281.063,-65.820,-176.721,6.961,148.335
C01114=1209.703,280.815,-65.791,-176.723,6.958,148.335
C01115=1209.707,280.567,-65.763,-176.725,6.956,148.335
C01116=1209.712,280.319,-65.735,-176.728,6.953,148.335
C01117=1209.716,280.070,-65.706,-176.731,6.951,148.335
C01118=1209.720,279.821,-65.678,-176.733,6.949,148.335
C01119=1209.725,279.573,-65.650,-176.736,6.946,148.335
C01120=1209.729,279.324,-65.621,-176.738,6.944,148.336
C01121=1209.733,279.077,-65.593,-176.741,6.941,148.336
C01122=1209.738,278.828,-65.564,-176.743,6.939,148.336
C01123=1209.742,278.580,-65.536,-176.746,6.937,148.336
C01124=1209.747,278.331,-65.507,-176.748,6.934,148.336
C01125=1209.751,278.084,-65.480,-176.750,6.931,148.336
C01126=1209.755,277.835,-65.451,-176.754,6.929,148.336
C01127=1209.760,277.587,-65.423,-176.756,6.927,148.336
C01128=1209.764,277.338,-65.395,-176.758,6.924,148.336
C01129=1209.769,277.090,-65.367,-176.761,6.922,148.337
C01130=1209.772,276.841,-65.339,-176.763,6.919,148.337
C01131=1209.777,276.593,-65.310,-176.766,6.916,148.337
C01132=1209.781,276.345,-65.282,-176.768,6.915,148.337
C01133=1209.786,276.096,-65.254,-176.771,6.912,148.337
C01134=1209.790,275.848,-65.226,-176.773,6.909,148.337
C01135=1209.794,275.600,-65.198,-176.776,6.907,148.338
C01136=1209.799,275.350,-65.170,-176.778,6.905,148.338
C01137=1209.804,275.103,-65.142,-176.781,6.902,148.338
C01138=1209.807,274.854,-65.114,-176.783,6.900,148.338
C01139=1209.812,274.606,-65.085,-176.786,6.897,148.338
C01140=1209.816,274.357,-65.057,-176.788,6.895,148.338
C01141=1209.820,274.109,-65.029,-176.791,6.893,148.338
C01142=1209.825,273.861,-65.001,-176.793,6.890,148.338
C01143=1209.830,273.612,-64.974,-176.796,6.888,148.339
C01144=1209.834,273.364,-64.946,-176.798,6.886,148.339
C01145=1209.838,273.115,-64.917,-176.801,6.883,148.339
C01146=1209.843,272.867,-64.889,-176.803,6.881,148.339
C01147=1209.847,272.619,-64.861,-176.806,6.878,148.339
C01148=1209.851,272.370,-64.834,-176.809,6.876,148.339
C01149=1209.856,272.122,-64.806,-176.811,6.874,148.339
C01150=1209.860,271.874,-64.778,-176.814,6.871,148.339
C01151=1209.864,271.626,-64.750,-176.816,6.869,148.340
C01152=1209.869,271.376,-64.722,-176.818,6.867,148.340
C01153=1209.874,271.128,-64.694,-176.821,6.864,148.340
C01154=1209.878,270.880,-64.666,-176.824,6.862,148.340
C01155=1209.882,270.631,-64.639,-176.826,6.860,148.340
C01156=1209.886,270.383,-64.611,-176.829,6.857,148.341
C01157=1209.891,270.134,-64.582,-176.831,6.855,148.341
C01158=1209.895,269.886,-64.555,-176.834,6.853,148.341
C01159=1209.900,269.638,-64.528,-176.836,6.850,148.341
C01160=1209.904,269.390,-64.499,-176.838,6.848,148.341
C01161=1209.908,269.141,-64.472,-176.841,6.846,148.341
C01162=1209.913,268.893,-64.444,-176.844,6.843,148.341
C01163=1209.917,268.644,-64.417,-176.846,6.841,148.342
C01164=1209.922,268.396,-64.389,-176.849,6.838,148.342
C01165=1209.926,268.148,-64.361,-176.852,6.836,148.342
C01166=1209.930,267.899,-64.334,-176.854,6.834,148.342
C01167=1209.934,267.651,-64.306,-176.857,6.831,148.342
C01168=1209.939,267.402,-64.279,-176.859,6.829,148.342
C01169=1209.944,267.153,-64.250,-176.861,6.827,148.342
C01170=1209.948,266.905,-64.223,-176.864,6.825,148.343
C01171=1209.953,266.657,-64.195,-176.867,6.822,148.343
C01172=1209.957,266.408,-64.168,-176.869,6.820,148.343
C01173=1209.961,266.160,-64.140,-176.871,6.818,148.343
C01174=1209.966,265.911,-64.113,-176.875,6.816,148.343
C01175=1209.970,265.664,-64.085,-176.877,6.813,148.344
C01176=1209.974,265.414,-64.058,-176.879,6.811,148.344
C01177=1209.979,265.166,-64.031,-176.882,6.808,148.344
C01178=1209.983,264.918,-64.003,-176.884,6.806,148.344
C01179=1209.988,264.670,-63.976,-176.887,6.804,148.344
C01180=1209.992,264.421,-63.948,-176.889,6.801,148.344
C01181=1209.996,264.172,-63.921,-176.892,6.800,148.345
C01182=1210.001,263.924,-63.894,-176.894,6.797,148.345
C01183=1210.005,263.675,-63.865,-176.897,6.795,148.345
C01184=1210.010,263.403,-63.835,-176.899,6.792,148.345
C01185=1210.015,263.130,-63.805,-176.903,6.790,148.345
C01186=1210.020,262.857,-63.776,-176.905,6.788,148.346
C01187=1210.025,262.585,-63.745,-176.908,6.785,148.346
C01188=1210.029,262.336,-63.717,-176.911,6.783,148.346
C01189=1210.034,262.088,-63.690,-176.913,6.780,148.346
C01190=1210.038,261.839,-63.663,-176.916,6.778,148.346
C01191=1210.042,261.591,-63.637,-176.918,6.776,148.346
C01192=1210.046,261.342,-63.609,-176.921,6.773,148.347
C01193=1210.051,261.094,-63.581,-176.923,6.771,148.347
C01194=1210.055,260.845,-63.554,-176.926,6.769,148.347
C01195=1210.060,260.597,-63.527,-176.928,6.767,148.347
C01196=1210.065,260.348,-63.500,-176.931,6.764,148.347
C01197=1210.069,260.100,-63.473,-176.933,6.762,148.347
C01198=1210.073,259.851,-63.445,-176.936,6.760,148.348
C01199=1210.078,259.603,-63.418,-176.939,6.757,148.348
C01200=1210.082,259.354,-63.391,-176.941,6.755,148.348
C01201=1210.087,259.106,-63.364,-176.943,6.753,148.348
C01202=1210.091,258.858,-63.337,-176.946,6.751,148.348
C01203=1210.096,258.609,-63.310,-176.949,6.748,148.349
C01204=1210.099,258.360,-63.282,-176.951,6.746,148.349
C01205=1210.104,258.112,-63.255,-176.954,6.744,148.349
C01206=1210.109,257.863,-63.228,-176.956,6.742,148.349
C01207=1210.113,257.615,-63.201,-176.959,6.739,148.349
C01208=1210.117,257.367,-63.175,-176.961,6.737,148.350
C01209=1210.122,257.118,-63.148,-176.964,6.735,148.350
C01210=1210.126,256.870,-63.120,-176.966,6.733,148.350
C01211=1210.131,256.621,-63.093,-176.969,6.731,148.350
C01212=1210.135,256.372,-63.066,-176.972,6.729,148.350
C01213=1210.139,256.124,-63.040,-176.974,6.727,148.351
C01214=1210.144,255.875,-63.012,-176.976,6.725,148.351
C01215=1210.148,255.627,-62.985,-176.979,6.722,148.351
C01216=1210.153,255.378,-62.958,-176.982,6.720,148.351
C01217=1210.157,255.130,-62.932,-176.984,6.718,148.351
C01218=1210.162,254.882,-62.905,-176.986,6.716,148.351
C01219=1210.166,254.633,-62.878,-176.990,6.713,148.352
C01220=1210.171,254.385,-62.851,-176.992,6.711,148.352
C01221=1210.175,254.137,-62.824,-176.994,6.709,148.352
C01222=1210.179,253.887,-62.798,-176.997,6.707,148.352
C01223=1210.184,253.638,-62.770,-177.000,6.704,148.352
C01224=1210.188,253.390,-62.744,-177.002,6.702,148.353
C01225=1210.192,253.142,-62.717,-177.004,6.700,148.353
C01226=1210.197,252.893,-62.690,-177.007,6.698,148.353
C01227=1210.201,252.645,-62.663,-177.010,6.695,148.353
C01228=1210.206,252.396,-62.636,-177.012,6.693,148.354
C01229=1210.211,252.147,-62.610,-177.015,6.691,148.354
C01230=1210.215,251.899,-62.584,-177.017,6.689,148.354
C01231=1210.219,251.651,-62.556,-177.020,6.687,148.354
C01232=1210.224,251.402,-62.529,-177.022,6.684,148.354
C01233=1210.228,251.154,-62.503,-177.025,6.682,148.355
C01234=1210.233,250.905,-62.477,-177.028,6.681,148.355
C01235=1210.237,250.657,-62.450,-177.030,6.678,148.355
C01236=1210.241,250.408,-62.423,-177.033,6.676,148.355
C01237=1210.246,250.159,-62.397,-177.035,6.674,148.355
C01238=1210.250,249.911,-62.370,-177.038,6.672,148.356
C01239=1210.255,249.662,-62.343,-177.040,6.670,148.356
C01240=1210.259,249.414,-62.317,-177.043,6.668,148.356
C01241=1210.264,249.165,-62.290,-177.046,6.665,148.356
C01242=1210.268,248.917,-62.263,-177.048,6.663,148.356
C01243=1210.272,248.668,-62.237,-177.050,6.661,148.357
C01244=1210.277,248.419,-62.211,-177.053,6.659,148.357
C01245=1210.281,248.171,-62.184,-177.055,6.657,148.357
C01246=1210.286,247.922,-62.158,-177.058,6.654,148.357
C01247=1210.290,247.674,-62.131,-177.061,6.652,148.358
C01248=1210.295,247.425,-62.104,-177.063,6.650,148.358
C01249=1210.299,247.176,-62.078,-177.066,6.648,148.358
C01250=1210.304,246.928,-62.051,-177.068,6.646,148.358
C01251=1210.308,246.680,-62.026,-177.071,6.643,148.359
C01252=1210.313,246.431,-61.999,-177.074,6.642,148.359
C01253=1210.317,246.183,-61.973,-177.076,6.639,148.359
C01254=1210.322,245.934,-61.946,-177.079,6.637,148.359
C01255=1210.326,245.686,-61.920,-177.081,6.635,148.359
C01256=1210.331,245.437,-61.893,-177.083,6.633,148.360
C01257=1210.335,245.189,-61.867,-177.086,6.631,148.360
C01258=1210.339,244.940,-61.841,-177.089,6.629,148.360
C01259=1210.344,244.691,-61.815,-177.091,6.627,148.360
C01260=1210.348,244.442,-61.788,-177.094,6.625,148.361
C01261=1210.353,244.193,-61.762,-177.096,6.623,148.361
C01262=1210.357,243.946,-61.736,-177.099,6.620,148.361
C01263=1210.362,243.697,-61.710,-177.102,6.618,148.361
C01264=1210.366,243.449,-61.683,-177.104,6.616,148.361
C01265=1210.370,243.200,-61.657,-177.107,6.614,148.362
C01266=1210.375,242.951,-61.631,-177.109,6.612,148.362
C01267=1210.379,242.702,-61.604,-177.111,6.610,148.362
C01268=1210.384,242.454,-61.579,-177.115,6.607,148.362
C01269=1210.388,242.205,-61.552,-177.117,6.606,148.363
C01270=1210.393,241.957,-61.526,-177.119,6.603,148.363
C01271=1210.397,241.708,-61.500,-177.122,6.601,148.363
C01272=1210.402,241.460,-61.473,-177.125,6.600,148.363
C01273=1210.406,241.211,-61.448,-177.127,6.597,148.364
C01274=1210.410,240.962,-61.422,-177.129,6.596,148.364
C01275=1210.415,240.713,-61.396,-177.133,6.593,148.364
C01276=1210.420,240.466,-61.369,-177.135,6.591,148.364
C01277=1210.424,240.217,-61.344,-177.137,6.589,148.365
C01278=1210.428,239.968,-61.318,-177.140,6.587,148.365
C01279=1210.433,239.719,-61.292,-177.142,6.585,148.365
C01280=1210.437,239.471,-61.265,-177.145,6.583,148.365
C01281=1210.442,239.223,-61.240,-177.148,6.580,148.366
C01282=1210.447,238.973,-61.213,-177.150,6.578,148.366
C01283=1210.451,238.725,-61.188,-177.153,6.576,148.366
C01284=1210.455,238.476,-61.162,-177.155,6.574,148.366
C01285=1210.460,238.228,-61.136,-177.158,6.573,148.367
C01286=1210.464,237.980,-61.110,-177.160,6.570,148.367
C01287=1210.469,237.730,-61.084,-177.163,6.569,148.367
C01288=1210.474,237.459,-61.056,-177.166,6.566,148.367
C01289=1210.479,237.188,-61.027,-177.169,6.564,148.368
C01290=1210.484,236.916,-60.999,-177.172,6.561,148.368
C01291=1210.488,236.644,-60.971,-177.174,6.559,148.368
C01292=1210.493,236.397,-60.945,-177.176,6.557,148.368
C01293=1210.498,236.148,-60.919,-177.179,6.555,148.369
C01294=1210.502,235.899,-60.893,-177.182,6.554,148.369
C01295=1210.507,235.651,-60.868,-177.184,6.551,148.369
C01296=1210.511,235.402,-60.842,-177.187,6.549,148.369
C01297=1210.515,235.153,-60.816,-177.190,6.547,148.370
C01298=1210.519,234.904,-60.790,-177.192,6.545,148.370
C01299=1210.524,234.656,-60.765,-177.194,6.543,148.370
C01300=1210.528,234.407,-60.739,-177.197,6.541,148.370
C01301=1210.533,234.158,-60.713,-177.200,6.539,148.371
C01302=1210.538,233.910,-60.688,-177.202,6.537,148.371
C01303=1210.543,233.661,-60.662,-177.205,6.535,148.371
C01304=1210.547,233.412,-60.636,-177.208,6.532,148.371
C01305=1210.552,233.164,-60.611,-177.210,6.531,148.372
C01306=1210.556,232.916,-60.585,-177.212,6.528,148.372
C01307=1210.560,232.667,-60.559,-177.215,6.527,148.372
C01308=1210.565,232.417,-60.534,-177.218,6.525,148.372
C01309=1210.569,232.169,-60.509,-177.220,6.523,148.373
C01310=1210.574,231.920,-60.483,-177.223,6.521,148.373
C01311=1210.578,231.672,-60.458,-177.225,6.519,148.373
C01312=1210.583,231.424,-60.432,-177.228,6.517,148.374
C01313=1210.587,231.175,-60.406,-177.230,6.515,148.374
C01314=1210.592,230.927,-60.381,-177.233,6.512,148.374
C01315=1210.596,230.678,-60.355,-177.236,6.510,148.374
C01316=1210.600,230.428,-60.330,-177.238,6.508,148.375
C01317=1210.605,230.180,-60.305,-177.241,6.507,148.375
C01318=1210.609,229.931,-60.279,-177.243,6.504,148.375
C01319=1210.614,229.683,-60.253,-177.246,6.503,148.375
C01320=1210.619,229.434,-60.228,-177.248,6.501,148.376
C01321=1210.623,229.185,-60.203,-177.251,6.499,148.376
C01322=1210.628,228.937,-60.177,-177.254,6.497,148.376
C01323=1210.632,228.688,-60.151,-177.256,6.495,148.376
C01324=1210.637,228.439,-60.126,-177.258,6.493,148.377
C01325=1210.641,228.191,-60.101,-177.261,6.491,148.377
C01326=1210.646,227.942,-60.075,-177.264,6.488,148.377
C01327=1210.651,227.694,-60.050,-177.266,6.486,148.377
C01328=1210.655,227.444,-60.025,-177.269,6.484,148.378
C01329=1210.659,227.196,-59.999,-177.272,6.483,148.378
C01330=1210.664,226.947,-59.974,-177.274,6.481,148.378
C01331=1210.668,226.698,-59.949,-177.277,6.479,148.379
C01332=1210.673,226.450,-59.924,-177.279,6.477,148.379
C01333=1210.677,226.201,-59.898,-177.282,6.475,148.379
C01334=1210.682,225.953,-59.873,-177.284,6.473,148.380
C01335=1210.686,225.704,-59.848,-177.287,6.471,148.380
C01336=1210.691,225.455,-59.823,-177.290,6.469,148.380
C01337=1210.696,225.206,-59.797,-177.292,6.467,148.380
C01338=1210.700,224.959,-59.773,-177.294,6.465,148.381
C01339=1210.704,224.709,-59.747,-177.297,6.463,148.381
C01340=1210.709,224.460,-59.722,-177.300,6.461,148.381
C01341=1210.714,224.212,-59.697,-177.303,6.459,148.382
C01342=1210.718,223.963,-59.671,-177.305,6.457,148.382
C01343=1210.722,223.714,-59.647,-177.308,6.455,148.382
C01344=1210.726,223.466,-59.621,-177.310,6.453,148.382
C01345=1210.732,223.217,-59.597,-177.313,6.451,148.383
C01346=1210.736,222.968,-59.571,-177.316,6.449,148.383
C01347=1210.741,222.719,-59.546,-177.318,6.448,148.383
C01348=1210.744,222.471,-59.521,-177.320,6.445,148.383
C01349=1210.750,222.222,-59.497,-177.323,6.444,148.384
C01350=1210.754,221.974,-59.471,-177.326,6.442,148.384
C01351=1210.759,221.725,-59.446,-177.328,6.440,148.384
C01352=1210.763,221.476,-59.422,-177.331,6.438,148.385
C01353=1210.768,221.227,-59.396,-177.334,6.436,148.385
C01354=1210.773,220.979,-59.372,-177.336,6.434,148.385
C01355=1210.776,220.730,-59.347,-177.338,6.432,148.385
C01356=1210.781,220.481,-59.322,-177.341,6.430,148.386
C01357=1210.786,220.232,-59.297,-177.344,6.428,148.386
C01358=1210.790,219.984,-59.272,-177.346,6.427,148.386
C01359=1210.794,219.735,-59.247,-177.349,6.424,148.387
C01360=1210.800,219.486,-59.222,-177.352,6.422,148.387
C01361=1210.804,219.238,-59.198,-177.354,6.420,148.387
C01362=1210.808,218.989,-59.172,-177.357,6.418,148.388
C01363=1210.813,218.740,-59.148,-177.360,6.416,148.388
C01364=1210.817,218.492,-59.123,-177.362,6.414,148.388
C01365=1210.822,218.243,-59.098,-177.365,6.413,148.389
C01366=1210.827,217.994,-59.073,-177.367,6.411,148.389
C01367=1210.831,217.745,-59.049,-177.370,6.409,148.389
C01368=1210.836,217.497,-59.023,-177.373,6.407,148.390
C01369=1210.840,217.248,-58.999,-177.375,6.405,148.390
C01370=1210.845,216.999,-58.974,-177.378,6.403,148.390
C01371=1210.850,216.750,-58.950,-177.380,6.401,148.390
C01372=1210.854,216.501,-58.925,-177.383,6.399,148.391
C01373=1210.858,216.253,-58.900,-177.385,6.398,148.391
C01374=1210.862,216.004,-58.875,-177.388,6.396,148.391
C01375=1210.867,215.755,-58.851,-177.391,6.394,148.392
C01376=1210.872,215.507,-58.827,-177.393,6.392,148.392
C01377=1210.876,215.258,-58.802,-177.396,6.390,148.392
C01378=1210.881,215.009,-58.777,-177.398,6.388,148.392
C01379=1210.886,214.760,-58.753,-177.401,6.386,148.393
C01380=1210.890,214.512,-58.727,-177.403,6.384,148.393
C01381=1210.894,214.263,-58.703,-177.406,6.382,148.393
C01382=1210.900,214.014,-58.678,-177.409,6.381,148.394
C01383=1210.903,213.765,-58.654,-177.411,6.379,148.394
C01384=1210.908,213.517,-58.629,-177.414,6.377,148.394
C01385=1210.913,213.268,-58.605,-177.417,6.375,148.395
C01386=1210.917,213.019,-58.580,-177.419,6.373,148.395
C01387=1210.922,212.770,-58.556,-177.422,6.371,148.395
C01388=1210.927,212.522,-58.531,-177.424,6.369,148.396
C01389=1210.931,212.273,-58.507,-177.427,6.367,148.396
C01390=1210.935,212.024,-58.483,-177.429,6.366,148.396
C01391=1210.940,211.775,-58.458,-177.432,6.364,148.397
C01392=1210.945,211.505,-58.432,-177.435,6.362,148.397
C01393=1210.950,211.234,-58.404,-177.438,6.359,148.397
C01394=1210.955,210.964,-58.379,-177.440,6.357,148.397
C01395=1210.960,210.694,-58.352,-177.444,6.356,148.398
C01396=1210.965,210.445,-58.328,-177.446,6.354,148.398
C01397=1210.969,210.196,-58.303,-177.448,6.352,148.399
C01398=1210.973,209.947,-58.279,-177.451,6.350,148.399
C01399=1210.978,209.699,-58.255,-177.454,6.348,148.399
C01400=1210.983,209.450,-58.230,-177.456,6.346,148.400
C01401=1210.987,209.201,-58.207,-177.459,6.345,148.400
C01402=1210.992,208.952,-58.182,-177.462,6.343,148.400
C01403=1210.996,208.703,-58.158,-177.464,6.341,148.401
C01404=1211.001,208.455,-58.134,-177.467,6.339,148.401
C01405=1211.006,208.206,-58.109,-177.470,6.337,148.401
C01406=1211.010,207.957,-58.085,-177.472,6.335,148.402
C01407=1211.014,207.708,-58.061,-177.475,6.334,148.402
C01408=1211.019,207.459,-58.037,-177.477,6.332,148.402
C01409=1211.024,207.211,-58.013,-177.480,6.330,148.403
C01410=1211.028,206.963,-57.989,-177.483,6.328,148.403
C01411=1211.033,206.713,-57.964,-177.485,6.326,148.403
C01412=1211.037,206.464,-57.940,-177.488,6.324,148.404
C01413=1211.042,206.216,-57.916,-177.490,6.322,148.404
C01414=1211.047,205.967,-57.891,-177.493,6.320,148.404
C01415=1211.052,205.718,-57.868,-177.495,6.319,148.404
C01416=1211.055,205.469,-57.844,-177.498,6.317,148.405
C01417=1211.060,205.221,-57.820,-177.501,6.315,148.405
C01418=1211.065,204.972,-57.795,-177.503,6.313,148.405
C01419=1211.070,204.723,-57.772,-177.505,6.312,148.406
C01420=1211.074,204.474,-57.748,-177.508,6.310,148.406
C01421=1211.079,204.225,-57.724,-177.511,6.308,148.406
C01422=1211.083,203.976,-57.700,-177.513,6.306,148.407
C01423=1211.088,203.727,-57.675,-177.516,6.305,148.407
C01424=1211.092,203.478,-57.652,-177.519,6.303,148.407
C01425=1211.097,203.230,-57.628,-177.521,6.301,148.408
C01426=1211.101,202.982,-57.604,-177.524,6.299,148.408
C01427=1211.106,202.733,-57.580,-177.527,6.297,148.408
C01428=1211.111,202.484,-57.556,-177.529,6.296,148.409
C01429=1211.116,202.235,-57.532,-177.532,6.294,148.409
C01430=1211.120,201.986,-57.508,-177.535,6.292,148.410
C01431=1211.124,201.737,-57.484,-177.537,6.290,148.410
C01432=1211.129,201.488,-57.460,-177.540,6.288,148.410
C01433=1211.133,201.239,-57.437,-177.543,6.286,148.411
C01434=1211.138,200.991,-57.413,-177.545,6.285,148.411
C01435=1211.142,200.742,-57.389,-177.547,6.284,148.411
C01436=1211.148,200.493,-57.365,-177.550,6.282,148.412
C01437=1211.152,200.244,-57.341,-177.553,6.280,148.412
C01438=1211.157,199.996,-57.317,-177.555,6.278,148.412
C01439=1211.161,199.747,-57.294,-177.558,6.276,148.413
C01440=1211.166,199.498,-57.270,-177.560,6.274,148.413
C01441=1211.170,199.248,-57.246,-177.563,6.273,148.413
C01442=1211.174,199.000,-57.222,-177.566,6.271,148.414
C01443=1211.179,198.751,-57.199,-177.568,6.269,148.414
C01444=1211.184,198.502,-57.175,-177.571,6.267,148.414
C01445=1211.188,198.254,-57.151,-177.574,6.265,148.415
C01446=1211.193,198.005,-57.128,-177.576,6.263,148.415
C01447=1211.197,197.756,-57.104,-177.578,6.262,148.415
C01448=1211.202,197.507,-57.081,-177.581,6.261,148.416
C01449=1211.207,197.258,-57.057,-177.584,6.259,148.416
C01450=1211.211,197.010,-57.033,-177.586,6.257,148.416
C01451=1211.216,196.761,-57.010,-177.589,6.255,148.417
C01452=1211.220,196.512,-56.986,-177.592,6.253,148.417
C01453=1211.225,196.263,-56.962,-177.594,6.251,148.417
C01454=1211.229,196.014,-56.939,-177.597,6.250,148.418
C01455=1211.234,195.765,-56.916,-177.600,6.248,148.418
C01456=1211.239,195.516,-56.892,-177.602,6.247,148.419
C01457=1211.243,195.268,-56.868,-177.604,6.245,148.419
C01458=1211.248,195.019,-56.845,-177.607,6.243,148.419
C01459=1211.253,194.770,-56.821,-177.610,6.241,148.420
C01460=1211.257,194.521,-56.798,-177.612,6.239,148.420
C01461=1211.262,194.272,-56.774,-177.615,6.238,148.420
C01462=1211.266,194.023,-56.751,-177.618,6.236,148.421
C01463=1211.271,193.774,-56.727,-177.620,6.234,148.421
C01464=1211.276,193.525,-56.704,-177.623,6.232,148.421
C01465=1211.280,193.276,-56.681,-177.625,6.231,148.422
C01466=1211.284,193.028,-56.657,-177.628,6.229,148.422
C01467=1211.289,192.779,-56.634,-177.630,6.227,148.422
C01468=1211.294,192.531,-56.611,-177.633,6.226,148.423
C01469=1211.299,192.282,-56.587,-177.636,6.224,148.423
C01470=1211.304,192.032,-56.564,-177.638,6.222,148.423
C01471=1211.308,191.783,-56.541,-177.641,6.220,148.424
C01472=1211.313,191.534,-56.517,-177.644,6.220,148.424
C01473=1211.318,191.285,-56.494,-177.646,6.218,148.425
C01474=1211.322,191.037,-56.471,-177.649,6.216,148.425
C01475=1211.326,190.788,-56.447,-177.651,6.214,148.425
C01476=1211.331,190.539,-56.424,-177.654,6.212,148.426
C01477=1211.335,190.290,-56.400,-177.657,6.210,148.426
C01478=1211.340,190.041,-56.377,-177.659,6.209,148.426
C01479=1211.345,189.793,-56.355,-177.662,6.208,148.427
C01480=1211.349,189.544,-56.331,-177.664,6.206,148.427
C01481=1211.354,189.295,-56.308,-177.667,6.204,148.428
C01482=1211.359,189.046,-56.285,-177.669,6.202,148.428
C01483=1211.363,188.797,-56.261,-177.672,6.200,148.428
C01484=1211.367,188.548,-56.238,-177.675,6.198,148.429
C01485=1211.372,188.299,-56.215,-177.677,6.197,148.429
C01486=1211.377,188.050,-56.192,-177.680,6.196,148.429
C01487=1211.382,187.801,-56.169,-177.683,6.194,148.430
C01488=1211.386,187.553,-56.147,-177.685,6.192,148.430
C01489=1211.391,187.304,-56.123,-177.688,6.190,148.431
C01490=1211.396,187.054,-56.100,-177.691,6.189,148.431
C01491=1211.400,186.806,-56.077,-177.693,6.187,148.431
C01492=1211.404,186.557,-56.054,-177.695,6.186,148.432
C01493=1211.410,186.308,-56.031,-177.698,6.184,148.432
C01494=1211.414,186.059,-56.008,-177.701,6.182,148.432
C01495=1211.418,185.811,-55.985,-177.703,6.180,148.433
C01496=1211.424,185.541,-55.960,-177.706,6.179,148.433
C01497=1211.429,185.271,-55.935,-177.709,6.177,148.434
C01498=1211.434,185.002,-55.910,-177.712,6.175,148.434
C01499=1211.439,184.732,-55.885,-177.714,6.173,148.434
C01500=1211.443,184.483,-55.862,-177.717,6.172,148.435
C01501=1211.448,184.234,-55.839,-177.720,6.170,148.435
C01502=1211.453,183.984,-55.816,-177.723,6.168,148.436
C01503=1211.457,183.736,-55.794,-177.725,6.167,148.436
C01504=1211.462,183.487,-55.771,-177.728,6.165,148.436
C01505=1211.467,183.238,-55.747,-177.730,6.164,148.437
C01506=1211.471,182.989,-55.725,-177.733,6.162,148.437
C01507=1211.476,182.741,-55.702,-177.736,6.160,148.437
C01508=1211.480,182.492,-55.680,-177.738,6.159,148.438
C01509=1211.485,182.242,-55.657,-177.740,6.157,148.438
C01510=1211.489,181.994,-55.634,-177.743,6.155,148.439
C01511=1211.494,181.745,-55.611,-177.746,6.154,148.439
C01512=1211.499,181.496,-55.588,-177.749,6.152,148.439
C01513=1211.503,181.247,-55.566,-177.751,6.151,148.440
C01514=1211.508,180.998,-55.542,-177.754,6.149,148.440
C01515=1211.513,180.749,-55.521,-177.756,6.147,148.441
C01516=1211.518,180.500,-55.497,-177.759,6.146,148.441
C01517=1211.522,180.251,-55.475,-177.761,6.145,148.441
C01518=1211.527,180.002,-55.452,-177.764,6.143,148.442
C01519=1211.531,179.754,-55.429,-177.766,6.141,148.442
C01520=1211.536,179.505,-55.406,-177.769,6.140,148.443
C01521=1211.540,179.255,-55.384,-177.772,6.138,148.443
C01522=1211.545,179.007,-55.361,-177.774,6.137,148.443
C01523=1211.550,178.758,-55.339,-177.777,6.135,148.444
C01524=1211.554,178.509,-55.316,-177.779,6.133,148.444
C01525=1211.559,178.260,-55.294,-177.782,6.131,148.444
C01526=1211.564,178.011,-55.271,-177.784,6.130,148.445
C01527=1211.568,177.762,-55.249,-177.787,6.129,148.445
C01528=1211.573,177.513,-55.225,-177.790,6.127,148.446
C01529=1211.578,177.264,-55.204,-177.793,6.125,148.446
C01530=1211.582,177.015,-55.181,-177.795,6.123,148.446
C01531=1211.587,176.766,-55.158,-177.797,6.122,148.447
C01532=1211.591,176.518,-55.136,-177.800,6.121,148.447
C01533=1211.596,176.268,-55.113,-177.803,6.119,148.448
C01534=1211.601,176.020,-55.091,-177.806,6.117,148.448
C01535=1211.605,175.771,-55.069,-177.808,6.116,148.449
C01536=1211.610,175.521,-55.046,-177.811,6.114,148.449
C01537=1211.615,175.273,-55.024,-177.813,6.113,148.449
C01538=1211.620,175.023,-55.001,-177.816,6.111,148.450
C01539=1211.624,174.775,-54.978,-177.818,6.110,148.450
C01540=1211.629,174.526,-54.957,-177.821,6.108,148.450
C01541=1211.634,174.276,-54.934,-177.824,6.107,148.451
C01542=1211.638,174.028,-54.911,-177.827,6.105,148.451
C01543=1211.642,173.779,-54.889,-177.829,6.104,148.452
C01544=1211.647,173.529,-54.867,-177.831,6.102,148.452
C01545=1211.652,173.281,-54.844,-177.834,6.100,148.452
C01546=1211.656,173.032,-54.822,-177.837,6.098,148.453
C01547=1211.662,172.783,-54.800,-177.839,6.098,148.453
C01548=1211.666,172.534,-54.777,-177.842,6.096,148.454
C01549=1211.670,172.285,-54.755,-177.845,6.094,148.454
C01550=1211.676,172.036,-54.733,-177.847,6.092,148.454
C01551=1211.680,171.787,-54.710,-177.849,6.091,148.455
C01552=1211.685,171.539,-54.689,-177.852,6.089,148.455
C01553=1211.689,171.289,-54.666,-177.855,6.088,148.456
C01554=1211.694,171.040,-54.644,-177.857,6.087,148.456
C01555=1211.699,170.791,-54.622,-177.860,6.085,148.457
C01556=1211.703,170.543,-54.600,-177.863,6.083,148.457
C01557=1211.707,170.294,-54.578,-177.865,6.081,148.457
C01558=1211.712,170.044,-54.555,-177.868,6.081,148.458
C01559=1211.717,169.795,-54.533,-177.870,6.079,148.458
C01560=1211.722,169.546,-54.511,-177.873,6.077,148.459
C01561=1211.726,169.298,-54.489,-177.876,6.075,148.459
C01562=1211.731,169.048,-54.466,-177.878,6.074,148.459
C01563=1211.736,168.800,-54.445,-177.881,6.073,148.460
C01564=1211.740,168.550,-54.423,-177.884,6.071,148.460
C01565=1211.745,168.302,-54.401,-177.886,6.070,148.461
C01566=1211.749,168.052,-54.379,-177.888,6.068,148.461
C01567=1211.755,167.803,-54.357,-177.891,6.067,148.461
C01568=1211.759,167.554,-54.335,-177.894,6.066,148.462
C01569=1211.764,167.305,-54.313,-177.896,6.064,148.462
C01570=1211.768,167.057,-54.290,-177.899,6.062,148.463
C01571=1211.773,166.808,-54.268,-177.902,6.060,148.463
C01572=1211.777,166.559,-54.246,-177.904,6.059,148.464
C01573=1211.782,166.310,-54.225,-177.907,6.058,148.464
C01574=1211.787,166.060,-54.202,-177.910,6.056,148.464
C01575=1211.792,165.812,-54.180,-177.912,6.055,148.465
C01576=1211.796,165.562,-54.158,-177.914,6.053,148.465
C01577=1211.801,165.314,-54.137,-177.917,6.052,148.466
C01578=1211.806,165.065,-54.115,-177.920,6.051,148.466
C01579=1211.810,164.816,-54.093,-177.922,6.049,148.467
C01580=1211.815,164.567,-54.071,-177.925,6.047,148.467
C01581=1211.819,164.318,-54.049,-177.927,6.046,148.467
C01582=1211.824,164.069,-54.027,-177.930,6.045,148.468
C01583=1211.829,163.820,-54.005,-177.933,6.043,148.468
C01584=1211.834,163.571,-53.984,-177.936,6.041,148.469
C01585=1211.839,163.322,-53.963,-177.938,6.040,148.469
C01586=1211.844,163.072,-53.940,-177.940,6.038,148.469
C01587=1211.849,162.824,-53.918,-177.943,6.037,148.470
C01588=1211.853,162.574,-53.896,-177.946,6.036,148.470
C01589=1211.858,162.326,-53.875,-177.948,6.034,148.471
C01590=1211.862,162.076,-53.853,-177.951,6.032,148.471
C01591=1211.867,161.828,-53.831,-177.953,6.032,148.472
C01592=1211.872,161.578,-53.810,-177.956,6.030,148.472
C01593=1211.876,161.329,-53.788,-177.959,6.028,148.472
C01594=1211.881,161.080,-53.766,-177.961,6.027,148.473
C01595=1211.886,160.832,-53.745,-177.964,6.026,148.473
C01596=1211.890,160.582,-53.723,-177.967,6.024,148.474
C01597=1211.894,160.334,-53.701,-177.969,6.023,148.474
C01598=1211.899,160.084,-53.680,-177.971,6.021,148.475
C01599=1211.904,159.836,-53.658,-177.974,6.020,148.475
C01600=1211.909,159.566,-53.635,-177.977,6.019,148.476
C01601=1211.914,159.297,-53.611,-177.980,6.017,148.476
C01602=1211.919,159.028,-53.588,-177.983,6.015,148.477
C01603=1211.925,158.759,-53.565,-177.985,6.014,148.477
C01604=1211.930,158.510,-53.543,-177.988,6.012,148.477
C01605=1211.933,158.261,-53.522,-177.990,6.011,148.478
C01606=1211.938,158.012,-53.501,-177.993,6.009,148.478
C01607=1211.943,157.763,-53.479,-177.996,6.008,148.479
C01608=1211.947,157.514,-53.457,-177.998,6.007,148.479
C01609=1211.953,157.265,-53.436,-178.001,6.005,148.480
C01610=1211.957,157.016,-53.414,-178.003,6.004,148.480
C01611=1211.962,156.767,-53.392,-178.006,6.003,148.481
C01612=1211.967,156.518,-53.371,-178.009,6.001,148.481
C01613=1211.972,156.269,-53.350,-178.011,6.000,148.481
C01614=1211.976,156.021,-53.329,-178.014,5.998,148.482
C01615=1211.980,155.771,-53.307,-178.017,5.997,148.482
C01616=1211.985,155.522,-53.286,-178.019,5.996,148.483
C01617=1211.991,155.273,-53.265,-178.022,5.994,148.483
C01618=1211.995,155.023,-53.243,-178.024,5.993,148.484
C01619=1211.999,154.775,-53.222,-178.027,5.991,148.484
C01620=1212.004,154.526,-53.201,-178.030,5.990,148.484
C01621=1212.009,154.277,-53.179,-178.032,5.989,148.485
C01622=1212.014,154.027,-53.158,-178.035,5.987,148.485
C01623=1212.018,153.779,-53.136,-178.038,5.985,148.486
C01624=1212.023,153.530,-53.115,-178.040,5.984,148.486
C01625=1212.028,153.281,-53.094,-178.042,5.983,148.487
C01626=1212.032,153.031,-53.072,-178.045,5.982,148.487
C01627=1212.037,152.782,-53.051,-178.048,5.980,148.488
C01628=1212.042,152.533,-53.030,-178.050,5.978,148.488
C01629=1212.046,152.285,-53.009,-178.053,5.978,148.489
C01630=1212.052,152.036,-52.988,-178.056,5.976,148.489
C01631=1212.056,151.786,-52.966,-178.058,5.975,148.489
C01632=1212.060,151.537,-52.945,-178.061,5.973,148.490
C01633=1212.066,151.288,-52.924,-178.063,5.972,148.490
C01634=1212.070,151.039,-52.903,-178.066,5.971,148.491
C01635=1212.076,150.790,-52.882,-178.068,5.969,148.491
C01636=1212.079,150.541,-52.860,-178.071,5.968,148.492
C01637=1212.084,150.292,-52.839,-178.074,5.966,148.492
C01638=1212.089,150.043,-52.818,-178.076,5.965,148.492
C01639=1212.094,149.794,-52.797,-178.079,5.964,148.493
C01640=1212.099,149.545,-52.776,-178.081,5.962,148.493
C01641=1212.103,149.295,-52.755,-178.084,5.961,148.494
C01642=1212.107,149.047,-52.734,-178.087,5.960,148.494
C01643=1212.113,148.797,-52.713,-178.089,5.958,148.495
C01644=1212.118,148.548,-52.692,-178.092,5.957,148.495
C01645=1212.122,148.300,-52.671,-178.095,5.956,148.496
C01646=1212.127,148.051,-52.650,-178.097,5.955,148.496
C01647=1212.132,147.801,-52.629,-178.099,5.953,148.497
C01648=1212.136,147.552,-52.607,-178.102,5.952,148.497
C01649=1212.141,147.303,-52.586,-178.105,5.950,148.498
C01650=1212.145,147.054,-52.566,-178.107,5.949,148.498
C01651=1212.151,146.805,-52.545,-178.110,5.948,148.499
C01652=1212.155,146.556,-52.523,-178.113,5.946,148.499
C01653=1212.160,146.307,-52.503,-178.115,5.945,148.499
C01654=1212.164,146.057,-52.482,-178.118,5.944,148.500
C01655=1212.169,145.808,-52.461,-178.120,5.943,148.500
C01656=1212.174,145.559,-52.440,-178.123,5.941,148.501
C01657=1212.178,145.311,-52.419,-178.126,5.939,148.501
C01658=1212.183,145.061,-52.398,-178.128,5.939,148.502
C01659=1212.188,144.813,-52.378,-178.131,5.937,148.502
C01660=1212.193,144.563,-52.357,-178.133,5.936,148.503
C01661=1212.197,144.314,-52.337,-178.136,5.934,148.503
C01662=1212.203,144.065,-52.316,-178.138,5.933,148.504
C01663=1212.208,143.816,-52.295,-178.141,5.932,148.504
C01664=1212.211,143.567,-52.273,-178.143,5.931,148.505
C01665=1212.217,143.318,-52.252,-178.146,5.929,148.505
C01666=1212.221,143.069,-52.232,-178.149,5.928,148.506
C01667=1212.225,142.820,-52.212,-178.151,5.927,148.506
C01668=1212.231,142.570,-52.191,-178.154,5.925,148.506
C01669=1212.235,142.321,-52.170,-178.157,5.924,148.507
C01670=1212.240,142.072,-52.149,-178.159,5.922,148.507
C01671=1212.245,141.823,-52.129,-178.162,5.922,148.508
C01672=1212.250,141.574,-52.108,-178.165,5.920,148.508
C01673=1212.254,141.325,-52.088,-178.167,5.919,148.509
C01674=1212.259,141.076,-52.067,-178.170,5.918,148.509
C01675=1212.264,140.827,-52.046,-178.172,5.917,148.510
C01676=1212.269,140.578,-52.025,-178.175,5.915,148.510
C01677=1212.273,140.329,-52.005,-178.177,5.914,148.511
C01678=1212.278,140.080,-51.984,-178.180,5.912,148.511
C01679=1212.283,139.830,-51.964,-178.183,5.911,148.512
C01680=1212.287,139.581,-51.943,-178.185,5.910,148.512
C01681=1212.293,139.332,-51.922,-178.188,5.908,148.513
C01682=1212.297,139.083,-51.902,-178.190,5.908,148.513
C01683=1212.302,138.834,-51.881,-178.193,5.906,148.514
C01684=1212.307,138.585,-51.860,-178.195,5.905,148.514
C01685=1212.311,138.336,-51.840,-178.198,5.903,148.515
C01686=1212.316,138.087,-51.820,-178.200,5.902,148.515
C01687=1212.321,137.838,-51.799,-178.204,5.901,148.516
C01688=1212.326,137.588,-51.779,-178.206,5.900,148.516
C01689=1212.330,137.339,-51.759,-178.208,5.898,148.516
C01690=1212.335,137.090,-51.738,-178.211,5.898,148.517
C01691=1212.340,136.841,-51.717,-178.214,5.896,148.517
C01692=1212.344,136.592,-51.697,-178.216,5.895,148.518
C01693=1212.349,136.343,-51.676,-178.219,5.893,148.518
C01694=1212.354,136.093,-51.656,-178.221,5.892,148.519
C01695=1212.358,135.844,-51.636,-178.224,5.891,148.519
C01696=1212.364,135.595,-51.615,-178.226,5.890,148.520
C01697=1212.368,135.346,-51.595,-178.229,5.888,148.520
C01698=1212.372,135.097,-51.574,-178.232,5.888,148.521
C01699=1212.377,134.848,-51.555,-178.234,5.886,148.521
C01700=1212.382,134.598,-51.534,-178.237,5.885,148.522
C01701=1212.387,134.350,-51.514,-178.240,5.883,148.522
C01702=1212.392,134.101,-51.493,-178.242,5.882,148.523
C01703=1212.397,133.852,-51.474,-178.245,5.881,148.523
C01704=1212.402,133.583,-51.451,-178.247,5.880,148.524
C01705=1212.407,133.314,-51.429,-178.250,5.879,148.524
C01706=1212.412,133.046,-51.407,-178.253,5.877,148.525
C01707=1212.417,132.777,-51.386,-178.255,5.876,148.525
C01708=1212.422,132.528,-51.365,-178.259,5.875,148.526
C01709=1212.426,132.279,-51.345,-178.261,5.874,148.526
C01710=1212.432,132.029,-51.325,-178.264,5.872,148.527
C01711=1212.437,131.781,-51.305,-178.266,5.871,148.527
C01712=1212.441,131.532,-51.284,-178.269,5.870,148.528
C01713=1212.446,131.282,-51.265,-178.271,5.869,148.528
C01714=1212.450,131.033,-51.244,-178.274,5.867,148.529
C01715=1212.455,130.784,-51.225,-178.277,5.867,148.529
C01716=1212.460,130.534,-51.204,-178.279,5.865,148.530
C01717=1212.465,130.285,-51.183,-178.282,5.864,148.530
C01718=1212.470,130.037,-51.164,-178.285,5.862,148.531
C01719=1212.474,129.788,-51.144,-178.287,5.861,148.531
C01720=1212.479,129.538,-51.124,-178.290,5.860,148.532
C01721=1212.484,129.289,-51.104,-178.292,5.859,148.532
C01722=1212.488,129.039,-51.084,-178.295,5.858,148.533
C01723=1212.493,128.790,-51.063,-178.297,5.857,148.533
C01724=1212.498,128.542,-51.043,-178.300,5.856,148.534
C01725=1212.503,128.292,-51.023,-178.303,5.854,148.534
C01726=1212.508,128.043,-51.003,-178.305,5.853,148.535
C01727=1212.512,127.794,-50.983,-178.308,5.852,148.535
C01728=1212.517,127.545,-50.963,-178.310,5.851,148.536
C01729=1212.522,127.296,-50.944,-178.313,5.849,148.536
C01730=1212.527,127.047,-50.924,-178.315,5.848,148.537
C01731=1212.531,126.798,-50.904,-178.318,5.847,148.537
C01732=1212.536,126.548,-50.884,-178.321,5.846,148.538
C01733=1212.541,126.299,-50.864,-178.323,5.845,148.538
C01734=1212.546,126.050,-50.844,-178.326,5.844,148.539
C01735=1212.550,125.801,-50.824,-178.328,5.843,148.539
C01736=1212.555,125.552,-50.804,-178.331,5.841,148.540
C01737=1212.560,125.302,-50.785,-178.333,5.840,148.540
C01738=1212.564,125.053,-50.764,-178.336,5.839,148.541
C01739=1212.570,124.804,-50.745,-178.339,5.838,148.541
C01740=1212.574,124.555,-50.725,-178.342,5.837,148.542
C01741=1212.579,124.306,-50.705,-178.344,5.836,148.542
C01742=1212.584,124.056,-50.685,-178.346,5.835,148.543
C01743=1212.589,123.808,-50.665,-178.349,5.833,148.543
C01744=1212.593,123.558,-50.646,-178.352,5.833,148.544
C01745=1212.598,123.309,-50.626,-178.354,5.831,148.544
C01746=1212.602,123.060,-50.606,-178.357,5.830,148.545
C01747=1212.608,122.811,-50.586,-178.360,5.828,148.545
C01748=1212.613,122.561,-50.567,-178.362,5.827,148.546
C01749=1212.617,122.312,-50.546,-178.364,5.827,148.546
C01750=1212.622,122.064,-50.527,-178.367,5.825,148.547
C01751=1212.627,121.814,-50.507,-178.370,5.824,148.547
C01752=1212.632,121.564,-50.488,-178.372,5.823,148.548
C01753=1212.636,121.316,-50.467,-178.375,5.822,148.548
C01754=1212.642,121.067,-50.448,-178.377,5.821,148.549
C01755=1212.646,120.817,-50.429,-178.380,5.820,148.549
C01756=1212.650,120.568,-50.409,-178.382,5.819,148.550
C01757=1212.656,120.319,-50.390,-178.386,5.817,148.550
C01758=1212.660,120.070,-50.370,-178.388,5.816,148.551
C01759=1212.665,119.820,-50.350,-178.391,5.815,148.552
C01760=1212.670,119.572,-50.331,-178.393,5.814,148.552
C01761=1212.675,119.322,-50.311,-178.396,5.813,148.553
C01762=1212.680,119.072,-50.291,-178.398,5.812,148.553
C01763=1212.684,118.824,-50.273,-178.401,5.811,148.554
C01764=1212.689,118.575,-50.252,-178.404,5.809,148.554
C01765=1212.693,118.325,-50.233,-178.406,5.809,148.555
C01766=1212.699,118.076,-50.213,-178.408,5.808,148.555
C01767=1212.704,117.827,-50.194,-178.412,5.806,148.556
C01768=1212.708,117.577,-50.174,-178.414,5.805,148.556
C01769=1212.713,117.329,-50.155,-178.416,5.805,148.557
C01770=1212.718,117.079,-50.136,-178.419,5.803,148.557
C01771=1212.723,116.830,-50.116,-178.422,5.802,148.558
C01772=1212.728,116.581,-50.097,-178.424,5.800,148.558
C01773=1212.733,116.331,-50.077,-178.427,5.800,148.559
C01774=1212.737,116.083,-50.058,-178.429,5.799,148.559
C01775=1212.742,115.834,-50.038,-178.432,5.797,148.560
C01776=1212.747,115.585,-50.019,-178.434,5.796,148.560
C01777=1212.752,115.335,-49.999,-178.437,5.795,148.561
C01778=1212.756,115.086,-49.980,-178.440,5.794,148.561
C01779=1212.761,114.837,-49.961,-178.442,5.794,148.562
C01780=1212.766,114.588,-49.941,-178.445,5.792,148.562
C01781=1212.771,114.339,-49.922,-178.447,5.791,148.563
C01782=1212.775,114.089,-49.903,-178.450,5.790,148.563
C01783=1212.780,113.839,-49.884,-178.453,5.789,148.564
C01784=1212.785,113.590,-49.864,-178.455,5.788,148.564
C01785=1212.789,113.341,-49.845,-178.458,5.786,148.565
C01786=1212.795,113.092,-49.826,-178.460,5.785,148.565
C01787=1212.800,112.843,-49.806,-178.463,5.785,148.566
C01788=1212.805,112.594,-49.787,-178.466,5.783,148.566
C01789=1212.809,112.345,-49.768,-178.468,5.782,148.567
C01790=1212.814,112.096,-49.749,-178.470,5.781,148.568
C01791=1212.819,111.846,-49.729,-178.473,5.780,148.568
C01792=1212.823,111.597,-49.710,-178.476,5.779,148.569
C01793=1212.828,111.348,-49.691,-178.478,5.779,148.569
C01794=1212.833,111.098,-49.672,-178.481,5.777,148.570
C01795=1212.838,110.849,-49.653,-178.483,5.776,148.570
C01796=1212.843,110.600,-49.634,-178.486,5.776,148.571
C01797=1212.847,110.351,-49.615,-178.489,5.774,148.571
C01798=1212.852,110.102,-49.595,-178.491,5.773,148.572
C01799=1212.857,109.853,-49.576,-178.494,5.771,148.572
C01800=1212.862,109.603,-49.558,-178.497,5.771,148.573
C01801=1212.867,109.354,-49.538,-178.499,5.770,148.573
C01802=1212.871,109.105,-49.519,-178.502,5.768,148.574
C01803=1212.876,108.856,-49.500,-178.504,5.767,148.574
C01804=1212.881,108.606,-49.481,-178.507,5.767,148.575
C01805=1212.886,108.357,-49.462,-178.510,5.765,148.576
C01806=1212.891,108.108,-49.443,-178.512,5.764,148.576
C01807=1212.895,107.859,-49.424,-178.515,5.764,148.577
C01808=1212.901,107.590,-49.404,-178.517,5.762,148.577
C01809=1212.906,107.322,-49.383,-178.520,5.762,148.578
